10:	IF ip_state = BYTE#3 THEN (* Bei IP_Control anmelden *)
		url_length := LEN(domain_copy);
		char_count := 17 + url_length; (* sendebuffer initialisieren *)
		FOR i := 0 TO char_count DO
			S_BUF.BUFFER[i] := BYTE#00;
		END_FOR;
		tid := UINT_TO_BYTE(BYTE_TO_UINT(tid) + UINT#1);
		S_BUF.BUFFER[01] := tid; (* Transaction ID lowbyte *)
		S_BUF.BUFFER[02] := BYTE#16#01; (* Flags: highbyte *)
		S_BUF.BUFFER[05] := BYTE#16#01; (* Questions: lowbyte *)
		i := url_length + 12;	(* den servernamen von hinten nach vorne bearbeiten *)
		char_count := 0;
		WHILE i > 12 DO
			char := CODE(STR:=domain_copy,POS:=i - 12);
			IF char = BYTE#46 THEN (* prüfe auf haupt/sub domänen namens-teiler "." *)
				S_BUF.BUFFER[i] := INT_TO_BYTE(char_count); (* anstelle des teilers "." wird die länge des erkannten haupt/sub domänennames eingetragen *)
				char_count := 0;
			ELSE
				S_BUF.BUFFER[i] := char; (* char in buffer eintragen *)
				char_count := char_count + 1; (* anzahl char zählen *)
			END_IF;
			i := i - 1;
		END_WHILE;
		S_BUF.BUFFER[i] := INT_TO_BYTE(char_count); (* längenangabe des ganz linken (ersten) domänennamens eintragen *)
		i := url_length + 15; (* position hinter dem servernamen *)
		S_BUF.BUFFER[i] := BYTE#01; (* Type: A Hostaddress lowbyte *)
		i := i + 2;
		S_BUF.BUFFER[i] := BYTE#01; (* Class: IN lowbyte *)
		i := i + 1;
		(* IP Datenverkehr einrichten *)
		IP_C.C_PORT := WORD#53; (* Portnummer eintragen *)
		IP_C.C_IP := IP4_DNS; (* IP eintragen *)
		IP_C.C_MODE := BYTE#1; (* Mode: UDP+AKTIV+PORT+IP *)
		IP_C.C_ENABLE := TRUE; (* Verbindungsaufbau freigeben *)
		IP_C.TIME_RESET := TRUE; (* Zeitueberwachung rücksetzen *)
		IP_C.R_OBSERVE  := TRUE; (* Datenempfang ueberwachen *)
		S_BUF.SIZE := INT_TO_UINT(i); (* sendelänge eintragen *)
		R_BUF.SIZE := UINT#0; (* Empfangslänge rücksetzen *)
		state := 30;

        		(*####################  DEBUG-MESSAGE  ###################################*)
        		(*IF _debug_enable THEN
            		LOG_CL.NEW_MSG := 'DNS: S10 SEND';
            		LOG_MSG();
        		END_IF;*)
        		(*########################################################################*)
	END_IF;

30:	IF IP_C.ERROR <> DWORD#00 THEN
		ERROR := IP_C.ERROR;
		state := 99;
        		(*####################  DEBUG-MESSAGE  ###################################*)
        		(*IF _debug_enable THEN
            		LOG_CL.NEW_MSG := 'DNS: S30 ERROR ~1';
            		LOG_CL.PRINTF[1]  := DWORD_TO_STRING(ERROR);
            		LOG_MSG();
        		END_IF;*)
        		(*########################################################################*)

	ELSIF (S_BUF.SIZE = UINT#0) AND (tid = R_BUF.BUFFER[1]) AND (R_BUF.SIZE >= INT_TO_UINT(34 + url_length)) THEN	(* prüfe ob antwort telegramm die richtige Transaction-ID und mindestlänge hat *)
		ERROR := BYTE_TO_DWORD(R_BUF.BUFFER[3] AND BYTE#2#0000_1111); (* prüfe Return code der Flags. 4 bits *)
		IF ERROR = DWORD#00 THEN
			anc := R_BUF.BUFFER[7]; (* Anzahl der Answer-RR *)
			IP_C.R_OBSERVE := FALSE; (* Datenempfang ueberwachen *)
			state := 40;
		ELSE
			state := 99;
		END_IF;
	END_IF;

40:	IF anc > 0 THEN
		anc := anc - 1;
		WHILE i < R_BUF.SIZE DO
			x := R_BUF.BUFFER[i];
			IF rr_stop = FALSE THEN
				IF x > BYTE#63 THEN (* zeiger auf namen *)
					i := i + 1;
					rr_stop := TRUE;
				ELSIF x= BYTE#0 THEN (* namens ende *)
					rr_stop := TRUE;
				ELSE
					i := i + x; (* namen *)
				END_IF;
				i := i + 1;
			ELSE
				rr_stop := FALSE;
				IF R_BUF.BUFFER[i+1] = BYTE#1 AND R_BUF.BUFFER[i+3] = BYTE#1 THEN (* Type A / Class IN *)
					i := i + 4;
					ttl_tmp := DWORD_OF_BYTE(R_BUF.BUFFER[i],R_BUF.BUFFER[i+1],R_BUF.BUFFER[i+2],R_BUF.BUFFER[i+3]); (* Time to live *)
					i := i + 6;
					IF ttl_tmp >= ttl_last THEN (* TTL ist länger *)
						ttl_last := ttl_tmp;
						IP4 := DWORD_OF_BYTE(R_BUF.BUFFER[i],R_BUF.BUFFER[i+1],R_BUF.BUFFER[i+2],R_BUF.BUFFER[i+3]); (* IP-Adresse *)
					END_IF;
					i := i + 4;
				ELSE
					i := i + 9;
					i := i + R_BUF.BUFFER[i] + 1; (* offset zu nächsten Block *)
				END_IF;
				EXIT;
			END_IF;
		END_WHILE;
	ELSE
		IF ttl_last > DWORD#0 THEN (* gültige RR mit IP gefunden *)
			DONE := TRUE;
            		(*####################  DEBUG-MESSAGE  ###################################*)
            		(*IF _debug_enable THEN
                			LOG_CL.NEW_MSG := 'DNS: S40 OK';
                			LOG_MSG();
            		END_IF;*)
            		(*########################################################################*)
		END_IF;
		state := 99;
	END_IF;

99:	R_BUF.SIZE := UINT#0; (* Empfangslänge rücksetzen *)
	ip_state := BYTE#4; (* Abmelden *)
	state := 00;

END_CASE;

activate_last := ACTIVATE; (* letzten Status sichern zur Flankenerkennung *)
IP_FIFO(FIFO:=IP_C.FIFO,STATE:=ip_state,ID:=ip_id); (* IP_FIFO *)

(* revision history

ks	18. oct. 2008	rev 1.0
	original version

ks	20. oct. 2009	rev 1.1
	unbenutzten code entfernt, all buffer base 0

ks	20. dec. 2010	rev 1.2
	parsing nach rfc1305
*)


(*----------------------------------------------------------------------------------------------------------------*)
(* Flags: 0x0100 (Standard query)                                                                                            *)
(* 0... .... .... .... = Response: Message is a query                                                                   *)
(* .000 0... ....  = Opcode: Standard query (0)                                                                          *)
(* .... ..0. .... .... = Truncated: Message is not truncated                                                          *)
(* .... ...1 .... .... = Recursion desired: Do query recursively                                                    *)
(* .... .... .0.. .... = Z: reserved (0)                                                                                                  *)
(* .... .... ...0 .... = Non-authenticated data OK: Non-authenticated data is unacceptable *)
(*-----------------------------------------------------------------------------------------------------------------*)

(*      0  1  2  3  4  5  6  7  8  9  0  1  2  3  4  5  *)
(*    +--+--+--+--+--+--+--+--+--+--+--+--+--+--+--+--+ *)
(*    |                      ID                       | idx: 0/1   *)
(*    +--+--+--+--+--+--+--+--+--+--+--+--+--+--+--+--+ *)
(*    |QR|   Opcode  |AA|TC|RD|RA|   Z    |   RCODE   | idx: 2/3   *)
(*    +--+--+--+--+--+--+--+--+--+--+--+--+--+--+--+--+ *)
(*    |                    QDCOUNT                    | idx: 4/5   *)
(*    +--+--+--+--+--+--+--+--+--+--+--+--+--+--+--+--+ *)
(*    |                    ANCOUNT                    | idx: 6/7   *)
(*    +--+--+--+--+--+--+--+--+--+--+--+--+--+--+--+--+ *)
(*    |                    NSCOUNT                    | idx: 8/9   *)
(*    +--+--+--+--+--+--+--+--+--+--+--+--+--+--+--+--+ *)
(*    |                    ARCOUNT                    | idx: 10/11 *)
(*    +--+--+--+--+--+--+--+--+--+--+--+--+--+--+--+--+ *)

(*
Errorcodes  Description	References 
000	No error. 		 	The request completed successfully.
001	Format error. 		The name server was unable to interpret the query. 
002	Server failure.  	The name server was unable to process this query due to a problem with the name server. 
003	Name Error. 	 	Meaningful only for responses from an authoritative name server, this code signifies that the domain name referenced in the query does not exist.
004	Not Implemented. 	The name server does not support the requested kind of query.
005	Refused. 			The name server refuses to perform the specified operation for policy reasons.
  						 For example, a name server may not wish to provide the information to the particular requester, or a name server may not wish to perform a particular operation (e.g., zone transfer) for particular data.
006	YXDomain.			Name Exists when it should not. 
007	YXRRSet. RR			Set Exists when it should not. 
008	NXRRSet. RR			Set that should exist does not. 
009	NotAuth.			Server Not Authoritative for zone. 
010	NotZone,			Name not contained in zone. 
255	Timeout				No Response  
   

beispiel einer DNS Request von google.at
ein request mit 3 Answer-Blocks


Domain Name System (response)
[Request In: 3]
[Time: 0.027533000 seconds]
Transaction ID: 0x5e1a
Flags: 0x8180 (Standard query response, No error)
1... .... .... .... = Response: Message is a response
.000 0... .... .... = Opcode: Standard query (0)
.... .0.. .... .... = Authoritative: Server is not an authority for domain
.... ..0. .... .... = Truncated: Message is not truncated
.... ...1 .... .... = Recursion desired: Do query recursively
.... .... 1... .... = Recursion available: Server can do recursive queries
.... .... .0.. .... = Z: reserved (0)
.... .... ..0. .... = Answer authenticated: Answer/authority portion was not authenticated
.... .... .... 0000 = Reply code: No error (0)
Questions: 1
Answer RRs: 3
Authority RRs: 0
Additional RRs: 0

Queries
google.at: type A, class IN
Name: google.at
Type: A (Host address)
Class: IN (0x0001)

Answers
google.at: type A, class IN, addr 72.14.221.104
Name: google.at
Type: A (Host address)
Class: IN (0x0001)
Time to live: 19 minutes, 9 seconds
Data length: 4
Addr: 72.14.221.104

google.at: type A, class IN, addr 66.249.93.104
Name: google.at
Type: A (Host address)
Class: IN (0x0001)
Time to live: 19 minutes, 9 seconds
Data length: 4
Addr: 66.249.93.104

google.at: type A, class IN, addr 216.239.59.104
Name: google.at
Type: A (Host address)
Class: IN (0x0001)
Time to live: 19 minutes, 9 seconds
Data length: 4
Addr: 216.239.59.104
*)
END_FUNCTION_BLOCK

(* POU IP_FIFO, ST *)
FUNCTION_BLOCK IP_FIFO
VAR_IN_OUT
	FIFO : IP_FIFO_DATA;
	ID : BYTE;
	STATE : BYTE;
END_VAR
VAR
	tmp : INT;

	(*LOG_MSG : LOG_MSG;
	_debug_enable : BOOL := TRUE;*)

END_VAR

(*	version 1.0	18. oct. 2008
	programmer 	ks
	tested BY		ks

	IP_FIFO ist ein Zusatzbaustein füR die Zugriffsverwaltung auf IP_CONTROL
*)
IF NOT FIFO.INIT THEN
	FIFO.INIT := TRUE;
	FIFO.NW := 1;
	FIFO.NR := 1;
	FIFO.EMPTY := TRUE;
	FIFO.FULL := FALSE;
	FIFO.TOP := 128; (* Arraygroesse 1 bis x *)
	FIFO.MAX_ID := BYTE#1; (* maximale anzahl von Anmeldungen einer ID *)
END_IF;

(* wenn keine ID vorhanden dann die naechste freie ID zuteilen *)
IF ID = BYTE#00 THEN
	IF FIFO.ID < INT_TO_BYTE(FIFO.TOP) THEN
		ID := USINT_TO_BYTE(BYTE_TO_USINT(FIFO.ID) + USINT#1); (* ID +1 *)
		FIFO.ID := ID; (* ID eintragen *)
	    	(*####################  DEBUG-MESSAGE  ###################################*)
	    	(*IF _debug_enable THEN
	      		LOG_CL.NEW_MSG := 'FIFO: NEW ID:~1';
	      		LOG_CL.PRINTF[1]  := BYTE_TO_STRING(ID);
	      		LOG_MSG();
	    	END_IF;*)
	    	(*########################################################################*)
	ELSIF STATE < BYTE#200 THEN
		(*####################  DEBUG-MESSAGE  ###################################*)
		(*IF _debug_enable THEN
			LOG_CL.NEW_MSG := 'FIFO: OVERFLOW ADD ID';
			LOG_MSG();
		END_IF;*)
		(*########################################################################*)

		(* sollte nie passieren ! -> es sind zuviele teilnehmer angemeldet *)
		(* es wird keine Nummer vergeben und alle anfragen werden negativ beantwortet *)
		STATE := BYTE#255;
		RETURN;
	END_IF;
END_IF;

IF STATE = BYTE#1 AND NOT FIFO.FULL THEN (* Anmelden *)
	(* nur eintragen wenn maximale anzahl nicht ueberschritten wurde *)
	tmp := BYTE_TO_INT(ID);
	IF FIFO.Y[tmp] < FIFO.MAX_ID THEN
		FIFO.Y[tmp] := USINT_TO_BYTE(BYTE_TO_USINT(FIFO.Y[tmp]) + USINT#1); (* IP_ID Zähler +1 *)
		tmp := FIFO.NW; (* geht bei mir leider nicht anders *)
		FIFO.X[tmp] := ID;
		IF FIFO.NW = FIFO.TOP THEN FIFO.NW := 1; ELSE FIFO.NW := FIFO.NW + 1; END_IF;
		FIFO.FULL := FIFO.NW = FIFO.NR;
		FIFO.EMPTY := FALSE;
		STATE := BYTE#2; (* weiterschalten auf "Warten auf Freigabe" *)
		(*####################  DEBUG-MESSAGE  ###################################*)
		(*IF _debug_enable THEN
			LOG_CL.NEW_MSG := 'FIFO: ADD ID:~1';
			LOG_CL.PRINTF[1]  := BYTE_TO_STRING(ID);
			LOG_MSG();
		END_IF;*)
		(*########################################################################*)

	END_IF;
END_IF;

IF STATE = BYTE#2 AND NOT FIFO.EMPTY THEN (* check current stack element *)
	tmp := FIFO.NR; (* geht bei mir leider nicht anders *)
	IF ID = FIFO.X[tmp] THEN
	STATE := BYTE#3; (* weiterschalten auf "Zugriffsfreigabe" *)
	END_IF;
END_IF;

IF STATE = BYTE#4 AND NOT FIFO.EMPTY THEN (* remove from stack *)
	tmp := FIFO.NR; (* geht bei mir leider nicht anders *)
	IF ID = FIFO.X[tmp] THEN
		tmp := BYTE_TO_INT(ID); (* geht bei mir leider nicht anders *)
		FIFO.Y[tmp] := USINT_TO_BYTE(BYTE_TO_USINT(FIFO.Y[tmp]) - USINT#1); (* ID Zähler -1 *)
		IF FIFO.NR = FIFO.TOP THEN FIFO.NR := 1; ELSE FIFO.NR := FIFO.NR + 1; END_IF;
		FIFO.EMPTY := FIFO.NR = FIFO.NW;
		FIFO.FULL := FALSE;
		(*####################  DEBUG-MESSAGE  ###################################*)
		(*IF _debug_enable THEN
			LOG_CL.NEW_MSG := 'FIFO: REMOVE ID:~1';
			LOG_CL.PRINTF[1]  := BYTE_TO_STRING(ID);
			LOG_MSG();
		END_IF;*)
		(*########################################################################*)
	END_IF;
	STATE := BYTE#5; (* "Remove done" *)
END_IF;

(* revision history
ks	18. oct. 2008	rev 1.0
	original version

*)
END_FUNCTION_BLOCK

(* POU IP4_DECODE, ST *)
FUNCTION IP4_DECODE : DWORD
VAR_INPUT
	str : STRING(15);
END_VAR
VAR
	pos: INT;
END_VAR

(*
version 1.1	10. mar 2009
programmer 	kurt
tested by		hugo

IP4_DECODE testet ob ein string eine gültige IPv4 Adresse enthält und gibt die 4 Bytes der IP Adresse als DWORD zurück.

*)
pos := FIND(str, '.');
WHILE pos > 0 DO
	IP4_DECODE := SHL(IP4_DECODE,8) OR STRING_TO_DWORD(LEFT(str,pos - 1));
	str := DELETE(str, pos, 1);
	pos := FIND(str, '.');
END_WHILE;
IP4_DECODE := SHL(IP4_DECODE,8) OR STRING_TO_DWORD(str);


(* revision history
hm		29. feb 2008	rev 1.0
	original version

hm	10. mar. 2009	rev 1.1
	new algorythm
*)
END_FUNCTION

(* POU IP_CONTROL, ST *)
FUNCTION_BLOCK IP_CONTROL
VAR_IN_OUT
	IP_C : IP_C; (* IP_Control Verwaltungsstruktur *)
	S_BUF : NETWORK_BUFFER; (* Externer Sendbuffer *)
	R_BUF : NETWORK_BUFFER; (* Externer Receivebuffer *)
END_VAR
VAR_INPUT
	IP : DWORD; (* IP Adresse *)
	PORT : WORD; (* Port Nummer *)
	TIME_OUT : TIME; (* Ueberwachungszeit Connect / Send / Receive *)
END_VAR
VAR
	c_time : UDINT; (* CONNECT-Time (Zeit bei nicht vorhandener Verbindung) *)
	s_time : UDINT; (* SEND-Time    (Zeit seit letzten Datensenden) *)
	r_time : UDINT; (* RECEIVE-Time (Zeit seit letztem Datenempfang) *)

	c_enable : BOOL; (* Connect: freigabe *)
	c_ip : DWORD; (* Connect: aktuelle IP-Adresse *)
	c_ip_str : STRING(15);
	c_port : WORD; (* Connect: aktuelle Port-Nummer *)
	c_mode : BYTE; (* Connect: aktueller Mode UDP/TCP...... *)
	c_status : BYTE; (* Connect: Status (Errorcode) *)
	c_ready : BOOL; (* Connect: Verbindung aufgebaut *)
	c_ready_old : BOOL; (* Connect: letzter Zustand von c_ready für Flankenauswertung *)

	s_total : INT; (* Send: Gesamtanzahl Bytes zum senden *)
	s_cur_pos : INT; (* Send: aktuelle Sendeposition *)
	s_cur_size : INT; (* Send: aktuelle Sendegroesse *)
	s_max_size : INT; (* Send: maximale Telegrammlänge fuer Senden *)
	s_active : BOOL; (* Send: Daten senden ist aktiv *)
	s_status : BYTE; (* Send: Status (Errorcodes) *)
	s_ip_str : STRING(15);
	s_ip_exist : BOOL;

	r_status : BYTE; (* Receive: Status (Errorcodes) *)
	r_count : INT; (* Receive: Anzahl empfangener Bytes *)
	r_offset : INT; (* Receive: aktuelle Position in externen Receivebuffer *)
	r_max_size : INT; (* Receive: groesse des externen Empfangbuffers*)

	new_connection : BOOL; (* Neue Verbindungsparameter vorhanden *)
	tx : DWORD; (* letzter zeitwert *)
	error_time : DWORD; (* aktueller Timeout-Wert *)

	state: BYTE; (* schrittmerker für connect *)
	bytes_received : DINT;
	udp_mode : BOOL;

	socket : T_HSOCKET;
	server : T_HSOCKET;
	fbCreate	: FB_SocketUdpCreate;
	fbConnect : FB_SocketConnect;
	fbClose : FB_SocketClose;
	fbSendTo : FB_SocketUdpSendTo;
	fbReceiveFrom : FB_SocketUdpReceiveFrom;
	fbSend : FB_SocketSend;
	fbReceive : FB_SocketReceive;
	fbListen : FB_SocketListen;
	fbAccept : FB_SocketAccept;
	nErrId : UDINT;
	Send_Busy : BOOL;
	Send_Error : BOOL;
	Send_ErrId : UDINT;

	IPCR : IP_CONTROL_RESET;

	(*LOG_MSG : LOG_MSG;
	_debug_enable : BOOL := TRUE;
	debug_index : INT;
	debug_ID : INT;
	debug_lasterror : DWORD;
	state_last : INT;
	debug_last_id : INT := 255;*)

END_VAR

VAR CONSTANT
	STOP : BYTE := 0;
	UDP_INIT : BYTE:= 31;
	UDP_INIT_WAIT : BYTE:= 32;
	TC_INIT : BYTE := 51;
	TC_CONNECT : BYTE:= 52;
	TS_INIT : BYTE:= 53;
	TS_LISTEN_WAIT : BYTE:= 54;
	TS_ACCEPT : BYTE:= 55;
	TS_ACCEPT_WAIT : BYTE:= 56;
	C_CLOSE : BYTE := 190;
	C_CLOSE_WAIT : BYTE:= 191;
	C_CLOSE2 : BYTE := 192;
	C_CLOSE_WAIT2 : BYTE:= 193;
	C_WAIT : BYTE := 200;
	C_REC : BYTE := 210;
	C_REC_WAIT : BYTE := 211;
	C_SND : BYTE := 220;
	C_SND_WAIT1 : BYTE := 221;
	C_SND_WAIT2 : BYTE := 222;
END_VAR

(*

version 1.7		30. may. 2011
programmer 		ks
tested by			ks

IP_CONTROL ist ein Wrapper-Baustein um eine Hersteller neutrale Schnittstelle zum Ethernet zu schaffen



TYP 	TCP / UDP 	Aktiv / Passiv 		Port-Nummer erforderlich 	IP-Adresse erforderlich
0 		TCP 		Aktiv 			Ja 						Ja
1 		UDP 		Aktiv 			Ja 						Ja
2 		TCP 		Passiv 			Ja 						Ja (Adresse des aktiven Partners)
3 		UDP 		Passiv 			Ja 						Ja (Adresse des aktiven Partners)
4 		TCP 		Passiv 			Ja 						Nein (beliebiger aktiver Partner wird akzeptiert)
5 		UDP 		Passiv 			Ja 						Nein (beliebiger aktiver Partner wird akzeptiert)

*)
(* Bei PLC reset oder Programm Download werden alle alten Verbindungen geschlossen *)
IPCR();
IF NOT IPCR.READY THEN RETURN; END_IF;

(*####################  DEBUG-MESSAGE  ###################################*)
(*IF _debug_enable THEN
	IF IP_C.FIFO.ID > BYTE#0 THEN (* nur wenn Teilnehmer ID's vorhanden sind *)
		debug_index := IP_C.FIFO.NR;
		debug_ID := BYTE_TO_INT(IP_C.FIFO.X[debug_index]);
	END_IF;
END_IF;*)
(*########################################################################*)

(* read system time *)
tx := T_PLC_MS();

IF IP_C.C_PORT = 0 THEN
	IP_C.C_PORT := PORT; (* uebergebenen PORT durch parametrierten PORT ersetzen *)
END_IF;
IF IP_C.C_IP = 0 AND IP_C.C_MODE < 4 THEN
	IP_C.C_IP := IP; (* uebergebene IP durch paramtrierte IP ersetzen *)
END_IF;

new_connection := c_ip <> IP_C.C_IP OR c_mode <> IP_C.C_MODE OR c_port <> IP_C.C_PORT; (* neue Verbindungs erwünscht ? *)
c_enable := IP_C.C_ENABLE AND NOT new_connection;

IF IP_C.C_ENABLE AND IP_C.ERROR = 0 AND state = STOP THEN (* Freigabe,kein Fehler,kein Socket offen *)
	c_ip   := IP_C.C_IP;
	c_mode := IP_C.C_MODE;
	c_port := IP_C.C_PORT;
	c_ip_str := IP4_TO_STRING(c_ip);
	udp_mode := C_MODE.0; (* Mode 1,3,5 = udp *)

	error_time := TIME_TO_DWORD(MAX(T#200ms,TIME_OUT));
	IP_C.TIME_RESET := TRUE; (* Alle Timer ruecksetzen *)
	r_max_size := SIZEOF(R_BUF.BUFFER);
	s_max_size := SIZEOF(S_BUF.BUFFER);

	IF udp_mode THEN (* Mode: 1,3,5 = UDP CLIENT/SERVER *)
		state := UDP_INIT;
	ELSIF c_mode = 0 THEN (* Mode: 0 = TCP CLIENT *)
		state := TC_INIT;
	ELSE
		state := TS_INIT; (* Mode: 2,4 = TCP SERVER *)
	END_IF;

	IF c_mode < 5 THEN (* Empfänger-IP vorgeben *)
		s_ip_str := c_ip_str;
		s_ip_exist := TRUE;
	ELSE
		s_ip_str := '';
		s_ip_exist := FALSE;
	END_IF;

    	(*####################  DEBUG-MESSAGE  ###################################*)
	(*IF _debug_enable THEN
		LOG_CL.NEW_MSG := 'IP_CON: MODE ~1 / IP ~2 / PORT ~3 /ID ~6';
		LOG_CL.PRINTF[1] := BYTE_TO_STRING(C_MODE);
		LOG_CL.PRINTF[2] := IP4_TO_STRING(c_ip);
		LOG_CL.PRINTF[3] := WORD_TO_STRING(c_port);
		LOG_CL.PRINTF[6] := INT_TO_STRING(debug_ID);
		LOG_MSG();
	END_IF;*)
	(*########################################################################*)

END_IF;

(*####################  DEBUG-MESSAGE  ###################################*)
(*IF  _debug_enable THEN
	IF state <> state_last THEN
		LOG_CL.NEW_MSG := 'IP_STEP ~1 -IP_ID ~6';
		LOG_CL.PRINTF[1] := BYTE_TO_STRING(state);
		LOG_CL.PRINTF[6] := INT_TO_STRING(debug_ID);
		LOG_MSG();
		state_last := state;
	END_IF;
END_IF;*)
(*########################################################################*)

(* ---------------------------------------------- *)

CASE state OF

UDP_INIT: (* UDP_CLIENT + SERVER *)
	(* 1. bei UDP-Client wird als lokalport 0 vorgegeben, damit das System automatisch einen freien lokalen Port sucht
	    2. bei UDP Server muss der gewüschte lokalport verwendet werden *)

	fbCreate(bExecute := FALSE);
	fbCreate(	bExecute := TRUE , sSrvNetId := '', sLocalHost := '', nLocalPort := SEL(c_mode = 1,c_port,0) , tTimeOut := TIME_OUT);
	fbCreate.bExecute := FALSE; (* vorbelegung *)
	state := UDP_INIT_WAIT;

UDP_INIT_WAIT:
	fbCreate();
	IF NOT fbCreate.bBusy THEN
		IF NOT fbCreate.bError THEN
			socket := fbCreate.hSocket;
			c_ready := TRUE; (* Connected *)
			state := C_WAIT;
		ELSE
			c_status := 1; (* FB_SocketUdpCreate failed *)
			nErrId := fbCreate.nErrId;
			state := C_CLOSE;
		END_IF;
	END_IF;

(* ---------------------------------------------- *)
TC_INIT: (* TCP-CLIENT (AKTIV) *)
	fbConnect(bExecute := FALSE);
	fbConnect(bExecute := TRUE, sSrvNetId := '', sRemoteHost := c_ip_str, nRemotePort := c_port, tTimeout := TIME_OUT);
	fbConnect.bExecute := FALSE; (* vorbelegung *)
	state := TC_CONNECT;

(* ---------------------------------------------- *)
TC_CONNECT:
	IF NOT c_enable OR c_status = 255 THEN (* keine freigabe oder connect timeout *)
		state := C_CLOSE;
	END_IF;

	fbConnect();
	IF NOT fbConnect.bBusy THEN
		IF fbConnect.bError THEN
			nErrID := fbConnect.nErrId;
			state :=TC_INIT; (* Nochmals versuchen *)
		ELSE
			socket := fbConnect.hSocket;
			c_ready := TRUE; (* Connected *)
			state := C_WAIT;
		END_IF;
	END_IF;
(* ---------------------------------------------- *)
TS_INIT: (* TCP-SERVER (PASSIV) *)
	fbListen(bExecute := FALSE);
	fbListen(bExecute := TRUE , sSrvNetId:= '' , sLocalHost:= '' , nLocalPort:= c_port , tTimeout:= TIME_OUT);
	fbListen.bExecute := FALSE;
	state := TS_LISTEN_WAIT;
(* ---------------------------------------------- *)
TS_LISTEN_WAIT:
	fbListen();
	IF NOT fbListen.bBusy THEN
		IF fbListen.bError THEN
			c_status := 3; (* FB_SocketListen failed *)
			nErrID := fbListen.nErrId;
			state := C_CLOSE;
		ELSE
			server := fbListen.hListener;
			state := TS_ACCEPT;
		END_IF;
	END_IF;
(* ---------------------------------------------- *)
TS_ACCEPT:
	fbAccept(bExecute := FALSE);
	fbAccept(bExecute := TRUE, sSrvNetId := '', hListener := server, tTimeout := TIME_OUT);
	fbAccept.bExecute := FALSE;
	state := TS_ACCEPT_WAIT;
(* ---------------------------------------------- *)
TS_ACCEPT_WAIT:
	fbAccept();
	IF NOT fbAccept.bBusy THEN

		state := TS_ACCEPT; (* vorbelegung  *)

		IF fbAccept.bError THEN
			c_status := 4; (* FB_SocketAccept failed *)
			nErrID := fbAccept.nErrId;
			state := C_CLOSE;
		ELSE (* no error *)
			IF fbAccept.bAccepted THEN
				socket := fbAccept.hSocket;
				IF socket.remoteAddr.sAddr  <> c_ip_str AND c_mode <> 4 THEN
					state := C_CLOSE; (* Remote ablehnen - Verbindung beenden *)
				ELSE
					state := C_WAIT;
					c_ready := TRUE; (* Connected *)
				END_IF;
			END_IF; (* fbAccept.bAccepted *)
		END_IF; (* NOT fbAccept.bError *)
	END_IF; (*  NOT fbAccept.bBusy *)
(* ---------------------------------------------- *)
C_CLOSE:
	c_ready := FALSE;
	IF socket.handle > 0 THEN
		fbClose(bExecute := FALSE );
		fbClose(bExecute := TRUE, sSrvNetId := '',	hSocket := socket);
		fbClose.bExecute := FALSE;
		state := C_CLOSE_WAIT;
	ELSE
		state:= C_CLOSE2;
	END_IF;

C_CLOSE_WAIT:
	fbClose();
	IF NOT fbClose.bBusy THEN
		socket := TCPADS_NULL_HSOCKET; (* Socket rücksetzen *)
		nErrId:= SEL(fbClose.bError,0,fbClose.nErrId);
		state:= C_CLOSE2;
	END_IF;

C_CLOSE2:
	IF server.handle > 0 THEN
		fbClose(bExecute := FALSE );
		fbClose(bExecute := TRUE, sSrvNetId := '',	hSocket := server);
		fbClose.bExecute := FALSE;
		state := C_CLOSE_WAIT2;
	ELSE
		state:= STOP;
	END_IF;

C_CLOSE_WAIT2:
	fbClose();
	IF NOT fbClose.bBusy THEN
		server := TCPADS_NULL_HSOCKET; (* Socket rücksetzen *)
		nErrId:= SEL(fbClose.bError,0,fbClose.nErrId);
		state:= STOP;
	END_IF;

(* ---------------------------------------------- *)

C_WAIT: (* Warten auf Anforderung für Beenden *)
	IF NOT c_enable OR NOT c_ready THEN
		state:= C_CLOSE;
	ELSIF S_BUF.SIZE > 0 AND IP_C.MAILBOX[2] = 0 AND s_ip_exist THEN
		state:= C_SND;
	ELSIF IP_C.MAILBOX[3] = 0 THEN
		state:= C_REC;
	END_IF;

(* ---------------------------------------------- *)

C_REC: (* Daten empfangen *)
	IF R_BUF.SIZE >= INT_TO_UINT(r_max_size) THEN
		R_BUF.SIZE := UINT#0;
		r_status := 254; (* Empfangsbuffer wegen Überlauf rückgesetzt *)
	END_IF;

	r_offset := SEL(udp_mode,UINT_TO_INT(R_BUF.SIZE),0);
	r_count := r_max_size - r_offset;
	bytes_received := 0;

	IF udp_mode THEN
		fbReceiveFrom(bExecute := FALSE );
		fbReceiveFrom(bExecute:= TRUE, sSrvNetId := '', hSocket:= socket, cbLen := r_count, pDest:= ADR(R_BUF.BUFFER), tTimeout:= TIME_OUT);
		fbReceiveFrom.bExecute := FALSE; (* Vorbelegung *)
	ELSE
		fbReceive(bExecute:= FALSE);
		fbReceive(bExecute:= TRUE, sSrvNetId := '' , hSocket:= socket , cbLen:= r_count, pDest:= ADR(R_BUF.BUFFER[r_offset]) , tTimeout:= TIME_OUT);
		fbReceive.bExecute:= FALSE;
	END_IF;
	state := C_REC_WAIT;

C_REC_WAIT:
	IF udp_mode THEN
		fbReceiveFrom(); (* UDP Mode *)
		IF NOT fbReceiveFrom.bBusy THEN
			IF NOT fbReceiveFrom.bError THEN
				IF fbReceiveFrom.nRecBytes > 0 THEN
					IF c_mode <> BYTE#5 AND fbReceiveFrom.sRemoteHost  <> c_ip_str THEN
						R_BUF.SIZE := UINT#0;
					ELSE
						bytes_received := fbReceiveFrom.nRecBytes;
						IF NOT s_ip_exist THEN
							s_ip_str := fbReceiveFrom.sRemoteHost;
							s_ip_exist := TRUE;
						END_IF;
					END_IF;
				END_IF;
				state := C_WAIT;
			ELSIF fbReceiveFrom.nErrId = 16#80072746 THEN (* Verbindung vom Remote beendet *)
				c_status := 253;
				c_ready := FALSE;
				state := C_WAIT;
			ELSE
				nErrId := fbReceiveFrom.nErrId;
				state := C_WAIT;
			END_IF;
		END_IF;
	ELSE
		fbReceive(); (* TCP Mode *)
		IF NOT fbReceive.bBusy THEN
			IF NOT fbReceive.bError THEN
				IF fbReceive.nRecBytes > 0 THEN
					bytes_received := fbReceive.nRecBytes;
				END_IF;
			ELSIF fbReceive.nErrId = 16#8004 THEN (* Verbindung vom Remote beendet *)
				c_status := 253;
				c_ready := FALSE;
			ELSE
				nErrId := fbReceive.nErrId;
			END_IF;
			state := C_WAIT;
		END_IF;
	END_IF;

	IF bytes_received > 0 THEN
		r_time := tx; (* Receive Timer ruecksetzen *)
		R_BUF.SIZE := INT_TO_UINT(r_offset + DINT_TO_UINT(bytes_received)); (* aktuelle buffersize eintragen *)
		IP_C.MAILBOX[1] := IP_C.MAILBOX[1] + 1; (* Receive Info *)
		IF IP_C.MAILBOX[1] = 0 THEN IP_C.MAILBOX[1] := 1; END_IF;
    		(*####################  DEBUG-MESSAGE  ###################################*)
		(*IF _debug_enable THEN
			LOG_CL.NEW_MSG := 'IP_REC DATA: POS: ~1 : SIZE: ~2 TOTAL ~3 -IP_ID ~6';
			LOG_CL.PRINTF[1] := INT_TO_STRING(r_offset);
			LOG_CL.PRINTF[2] := INT_TO_STRING(r_count);
			LOG_CL.PRINTF[3] := UINT_TO_STRING(R_BUF.SIZE);
			LOG_CL.PRINTF[6] := INT_TO_STRING(debug_ID);
			LOG_MSG();
		END_IF;*)
		(*########################################################################*)
	END_IF;

(* ---------------------------------------------- *)
C_SND:
	IF S_BUF.SIZE > 0 THEN
		IF c_ready AND c_enable THEN
			IF NOT s_active THEN
				s_total := LIMIT(0,UINT_TO_INT(S_BUF.SIZE),r_max_size); (* Gesamtanzahl an Bytes limitieren und uebergeben *)
				s_cur_pos  := 0;
				s_cur_size := 0;
				s_active := TRUE; (* Sende-Betrieb aktivieren *)
			END_IF;

			s_cur_pos := s_cur_pos + s_cur_size; (* neue Sende-Datenposition bestimmen *)
			IF s_total > s_cur_pos THEN (* weitere Daten zum senden vorhanden ? *)
				s_cur_size := s_total - s_cur_pos;
				s_cur_size := LIMIT(0, s_cur_size, s_max_size); (* Telegrammlänge begrenzen *)
				s_time := tx; (* Send Timer ruecksetzen *)
				r_time := tx; (* Receive Timer ruecksetzen *)
				state := C_SND_WAIT1;
			ELSE (* keine weitere Sendedaten vorhanden -> Senden beenden *)
				s_active := FALSE;
				S_BUF.SIZE := 0;
				state := C_WAIT;
			END_IF;
		END_IF;
	END_IF;

C_SND_WAIT1:
	IF udp_mode THEN
		fbSendTo(bExecute := FALSE );
		fbSendTo(bExecute := TRUE, sSrvNetId := '', hSocket := socket , cbLen := s_cur_size, pSrc := ADR(S_BUF.BUFFER[s_cur_pos]), sRemoteHost := s_ip_str, nRemotePort := c_port, tTimeout:= TIME_OUT);
		fbSendTo.bExecute := FALSE;
	ELSE
		fbSend(bExecute := FALSE);
		fbSend(bExecute := TRUE, sSrvNetId := '', hSocket := socket , cbLen:= s_cur_size, pSrc:=ADR(S_BUF.BUFFER[s_cur_pos]), tTimeout:= TIME_OUT);
		fbSend.bExecute := FALSE;
	END_IF;
	state := C_SND_WAIT2;

C_SND_WAIT2:
	IF udp_mode THEN
		fbSendTo();
		Send_Busy := fbSendTo.bBusy;
		Send_Error := fbSendTo.bError;
		Send_ErrId := fbSendTo.nErrId;
	ELSE
		fbSend();
		Send_Busy := fbSend.bBusy;
		Send_Error := fbSend.bError;
		Send_ErrId := fbSend.nErrId;
	END_IF;

	IF NOT Send_Busy THEN
		IF NOT Send_Error THEN
    			(*####################  DEBUG-MESSAGE  ###################################*)
			(*IF _debug_enable THEN
				LOG_CL.NEW_MSG := 'IP_SEN SEND_COUNT ~1 -IP_ID ~6';
				LOG_CL.PRINTF[1] := DINT_TO_STRING(s_cur_size);
				LOG_CL.PRINTF[6] := INT_TO_STRING(debug_ID);
				LOG_MSG();
			END_IF;*)
			(*########################################################################*)
			state := C_SND;
		ELSE
			nErrId := Send_ErrId;
			state := C_WAIT;
    			(*####################  DEBUG-MESSAGE  ###################################*)
			(*IF _debug_enable THEN
				LOG_CL.NEW_MSG := 'IP_SEN SEND ERROR ~1 -IP_ID ~6';
				LOG_CL.PRINTF[1] := UDINT_TO_STRING(nErrId);
				LOG_CL.PRINTF[6] := INT_TO_STRING(debug_ID);
				LOG_MSG();
			END_IF;*)
			(*########################################################################*)
		END_IF;
	END_IF;

END_CASE;

(* ---------------------------------------------- *)

IF c_ready THEN
	IF NOT c_ready_old THEN (* Verbindung aufgebaut - positive Flanke erkannt *)
		IP_C.C_STATE := 254;
		IP_C.TIME_RESET := TRUE; (* Alle Timer ruecksetzen *)
    		(*####################  DEBUG-MESSAGE  ###################################*)
		(*IF _debug_enable THEN
			LOG_CL.NEW_MSG := 'IP_CON: CONNECTED -IP_ID ~6';
			LOG_CL.PRINTF[6] := INT_TO_STRING(debug_ID);
			LOG_MSG();
		END_IF;*)
		(*########################################################################*)
	ELSE
		IP_C.C_STATE := 255; (* Verbindung ist aufgebaut *)
	END_IF;
ELSE
	IF c_ready_old THEN (* Verbindung abgebaut - negative Flanke erkannt *)
		IP_C.C_STATE := 1;
		IP_C.MAILBOX[1] := 0; (* Receive Info rücksetzen *)
		IP_C.MAILBOX[2] := 0; (* Send-Pause rücksetzen *)
		IP_C.MAILBOX[3] := 0; (* Receive-Pause rücksetzen *)
		IF NOT new_connection THEN
			s_active := FALSE; (* Sendeaktivitäten stoppen *)
			S_BUF.SIZE := 0; (* Sendelänge löschen *)
			(*IP_C.TIME_RESET := TRUE; *) (* Alle Timer ruecksetzen *)
		END_IF;
    		(*####################  DEBUG-MESSAGE  ###################################*)
		(*IF _debug_enable THEN
			LOG_CL.NEW_MSG := 'IP_CON: DISCONNECTED';
			LOG_MSG();
		END_IF;*)
		(*########################################################################*)

	ELSE
		IP_C.C_STATE := 0; (* Verbindung ist abgebaut *)
	END_IF;
END_IF;

c_ready_old := c_ready;

(* ---------------------------------------------- *)

IF IP_C.TIME_RESET THEN (* Alle Timer ruecksetzen *)
	IP_C.TIME_RESET := FALSE; (* Reset rücksetzen *)
	c_time := tx; (* Connect Timer ruecksetzen *)
	s_time := tx; (* Send Timer ruecksetzen *)
	r_time := tx; (* Receive Timer ruecksetzen *)

	c_status := BYTE#0; (* letzten Connect Fehler rücksetzen *)
	s_status := BYTE#0; (* letzten Send Fehler rücksetzen *)
	r_status := BYTE#0; (* letzten Receive Fehler rücksetzen *)
END_IF;

IF IP_C.R_OBSERVE = FALSE THEN
    r_time := tx;
END_IF;

IF c_status = 0 AND tx - c_time > error_time AND c_enable AND NOT c_ready AND c_mode < 2 THEN (* Connect Timeout *)
	c_status := 255; (* Timeout-Fehler ausgeben *)
END_IF;
IF s_status = 0 AND tx - s_time > error_time AND s_active THEN (* Send Timeout *)
	s_status := 255; (* Timeout-Fehler ausgeben *)
END_IF;
IF r_status = 0 AND tx - r_time > error_time AND c_ready AND IP_C.R_OBSERVE THEN (* Receive Timeout *)
	r_status := 255; (* Timeout-Fehler ausgeben *)
END_IF;

IP_C.ERROR := DWORD_OF_BYTE(c_status,s_status,r_status,0);

(*####################  DEBUG-MESSAGE  ###################################*)
(*IF  _debug_enable THEN
	IF (IP_C.ERROR <> debug_lasterror) THEN
		LOG_CL.NEW_MSG := 'IP_ERROR ~1 -IP_ID ~6';
		LOG_CL.PRINTF[1] := DWORD_TO_STRING(IP_C.ERROR);
		LOG_CL.PRINTF[6] := INT_TO_STRING(debug_ID);
		LOG_MSG();

		debug_lasterror := IP_C.ERROR;
		debug_last_id := debug_ID;
	END_IF;
END_IF;*)
(*########################################################################*)

(* revision history
ks	18. oct. 2008	rev 1.0
	original version
ks	05. jan. 2009	rev 1.1
	zusätzlichen Parameter "Port" hinzugefügt, und Code bei Verbindungsaufbau angepasst
ks	28. feb. 2009	rev 1.2
	connect code angepasst und verkürzung der zyklen bei Send
ks	20. oct. 2009	rev 1.3
	network_buffer basis 0
ks	06. dec. 2009	rev 1.4
	receive_count MAILBOX[1]
ks	10. nov. 2010	rev 1.5
	send_pause MAILBOX[2] and receive_pause MAILBOX[3] 
ks	07. feb. 2011	rev 1.6
	Fehlercode 253 bei Remote-Verbindungsabbruch 
ks	30. may. 2011	rev 1.7
	Fehler bei Empfangsüberwachung
*)
END_FUNCTION_BLOCK

(* POU IP_CONTROL_RESET, ST *)
FUNCTION_BLOCK IP_CONTROL_RESET
VAR_INPUT
END_VAR
VAR_OUTPUT
	READY : BOOL;
END_VAR
VAR
	fbSocketCloseAll : FB_SocketCloseAll;
	step : BYTE;
END_VAR
(* On PLC reset or program download close all old connections *)

CASE TCP_SERVER_RESET OF

2:	READY := TRUE;
	RETURN;

1:	IF step = 0 THEN
		RETURN;
	END_IF;

0:	TCP_SERVER_RESET := 1; (* Reset ist aktiv *)
	step := 1;

END_CASE;

CASE step OF

0:	RETURN;

1:	fbSocketCloseAll(sSrvNetId:= '', bExecute:= TRUE, tTimeout:= T#10s );
	step := 2;

2:	fbSocketCloseAll(bExecute:= FALSE);
	IF fbSocketCloseAll.bBusy = FALSE THEN
		step := 0;
		TCP_SERVER_RESET := 2; (* Reset durchgeführt , Bereit zur Verwendung *)
	END_IF;

END_CASE;
END_FUNCTION_BLOCK

(* POU IP4_TO_STRING, ST *)
FUNCTION IP4_TO_STRING : STRING(15)
VAR_INPUT
	IP4 : DWORD;
END_VAR
VAR
	tmp : STRING(3);
END_VAR

(*
version 1.1	10. mar. 2009
programmer 	kurt
tested by	hugo

IP4_TO_STRING erzeugt eine IP Adresse als String aus einem DWORD..

*)
(* mask bits AND INSERT AT given position *)
tmp := BYTE_TO_STRING(DWORD_TO_BYTE(IP4));
IP4_TO_STRING := CONCAT('...', tmp);
tmp := BYTE_TO_STRING(DWORD_TO_BYTE(SHR(IP4,8)));
IP4_TO_STRING := INSERT(IP4_TO_STRING, tmp, 2);
tmp := BYTE_TO_STRING(DWORD_TO_BYTE(SHR(IP4,16)));
IP4_TO_STRING := INSERT(IP4_TO_STRING, tmp, 1);
tmp := BYTE_TO_STRING(DWORD_TO_BYTE(SHR(IP4,24)));
IP4_TO_STRING := CONCAT(tmp, IP4_TO_STRING);



(* revision history
hm	22. apr 2008	rev 1.0
	original version

hm	10. mar. 2009	rev 1.1
	improved code
*)
END_FUNCTION

(* POU STRING_TO_URL, ST *)
FUNCTION STRING_TO_URL : URL
VAR_INPUT
	STR : STRING(STRING_LENGTH);
	DEFAULT_PROTOCOL : STRING(10);
	DEFAULT_PATH : STRING(80);
END_VAR
VAR
	pos: INT;
	pos2: INT;
END_VAR
VAR_TEMP
	x : STRING(STRING_LENGTH);
END_VAR

(*
version 1.1	20. dec. 2010
programmer 	hugo
tested by		oscat

URL splits a unifrom resource locator in its conponents.

*)
(*

http://hans:geheim@www.example.org:80/demo/example.cgi?land=de&stadt=aa#abschnitt1
|       |      |         |         |   |                   |               |
|       |      |         Host      |   Pfad                Query           Anker
|       |      Passwort            Port
|       Benutzer
Protokoll

*)

(* check if string is empty and return empty url *)
IF STR = '' THEN RETURN; END_IF;

(* extract the protocol *)
(* first we check if the optional protocol is specified ending with a :// *)
pos := FIND(STR, '://');
IF pos > 0 THEN
	(* store protocol and restore the rest of url in temp *)
	STRING_TO_URL.PROTOCOL := LEFT(STR, pos - 1);
	x := RIGHT(STR, LEN(STR) - pos - 2);
ELSE
	x := STR;
	STRING_TO_URL.PROTOCOL := DEFAULT_PROTOCOL;
END_IF;

(* extract user and password if present ending with a @ *)
pos := FIND(x, '@');
IF pos > 0 THEN
	(* extract user *)
	pos2 := FIND(x,':')+1;
	IF pos2 > 1 AND pos2 <= pos THEN
		STRING_TO_URL.USER := LEFT(x,pos2 - 2);
		STRING_TO_URL.PASSWORD := MID(x, pos - pos2, pos2);
	ELSE
		STRING_TO_URL.USER := LEFT(x, pos - 2);
		STRING_TO_URL.PASSWORD := '';
	END_IF;
	x := RIGHT(x, LEN(x) - pos);
ELSE
	STRING_TO_URL.USER := '';
	STRING_TO_URL.PASSWORD := '';
END_IF;

(* extract anchor *)
pos := FIND(x, '#');
IF pos > 0 THEN
	STRING_TO_URL.ANCHOR := RIGHT(x, LEN(x) - pos);
	x := LEFT(x, pos - 1);
ELSE
	STRING_TO_URL.ANCHOR := '';
END_IF;

(* extract query  *)
pos := FIND(x, '?');
IF pos > 0 THEN
	STRING_TO_URL.QUERY := RIGHT(x, LEN(x) - pos);
	x := LEFT(x, pos - 1);
ELSE
	STRING_TO_URL.QUERY := '';
END_IF;

(* extract path  *)
pos := FIND(x, '/');
IF pos > 0 THEN
	STRING_TO_URL.PATH := RIGHT(x, LEN(x) - pos + 1);
	x := LEFT(x, pos - 1);
ELSE
	STRING_TO_URL.PATH := DEFAULT_PATH;
END_IF;

(* extract port and leave domain *)
pos := FIND(x, ':');
IF pos > 0 THEN
	STRING_TO_URL.PORT := STRING_TO_WORD(RIGHT(x, LEN(x) - pos));
	STRING_TO_URL.DOMAIN := LEFT(x, pos - 1);
ELSE
	STRING_TO_URL.PORT := 0;
	STRING_TO_URL.DOMAIN := x;
END_IF;

(* revision history
hm		18. apr 2008	rev 1.0
	original version

ks		20. dec. 2010	rev 1.1
	stringlength 250 , var x

*)
END_FUNCTION

(* POU FILE_PATH_SPLIT, ST *)
FUNCTION FILE_PATH_SPLIT : BOOL
VAR_INPUT
	FILENAME : STRING(STRING_LENGTH);
END_VAR
VAR_IN_OUT
	X : FILE_PATH_DATA;
END_VAR
VAR
	b : INT;
	c : INT;
	d : STRING(1);
	p1 : INT;
	p2 : INT;
END_VAR

(*
version 1.0		01. jan. 2011
programmer		ks
tested by			ks

FILE_PATH_SPLIT zerlegt einen Dateipfad in einzelne Elemente und legt diese in einer Datenstruktur ab.
*)
X.DRIVE := '';
X.DIRECTORY := '';
X.FILENAME := '';
c := LEN(FILENAME);
IF c = 0 THEN
	FILE_PATH_SPLIT := FALSE;
	RETURN;
END_IF;

FOR b := 1 TO c DO
	d := MID(FILENAME, 1, b);
	IF d = ':' THEN
		p1 := b;
	ELSIF d = '/' OR d = '\' THEN
		p2 := b;
	END_IF;
END_FOR;

IF p1 = 2 THEN
	X.DRIVE := LEFT(FILENAME,p1);
END_IF;

IF p2 > 0 AND p2 > p1 THEN
	X.DIRECTORY := MID(FILENAME,p2 - p1,p1+1); (* len , pos *)
END_IF;

X.FILENAME := RIGHT(FILENAME,c - MAX (p1,p2));
FILE_PATH_SPLIT := TRUE;

(* revision history
ks	01. jan. 2011	rev 1.0
	original version
*)
END_FUNCTION

(* POU ELEMENT_GET, ST *)
FUNCTION ELEMENT_GET : STRING(ELEMENT_LENGTH)
VAR_INPUT
	SEP : BYTE;
	POS : INT;
END_VAR
VAR_IN_OUT
	ELEMENT : STRING(ELEMENT_LENGTH);
END_VAR
VAR
	i : INT := 1;
	o : INT := 1;
	pt : POINTER TO ARRAY[1..ELEMENT_LENGTH] OF BYTE;
	po : POINTER TO ARRAY[1..ELEMENT_LENGTH] OF BYTE;
	cnt: INT;
	c: BYTE;
END_VAR

(*
version 1.0	05. apr. 2011
programmer 	ks
tested by		kst

ELEMENT_GET liefert das element an der stelle pos einer liste.
die liste liegt als string von elementen vor die mit den zeichen SEP separiert sind.

*)
(* load pointers *)
pt := ADR(ELEMENT);
po := ADR(ELEMENT_GET);

(* search for the n-th occurence of a separation character and store position in i *)
WHILE (cnt < pos) AND (i < ELEMENT_LENGTH) AND (pt^[i] > 0) DO
	IF pt^[i] = sep THEN cnt := cnt + 1; END_IF;
	i := i + 1;
END_WHILE;

(* copy the list element to output *)
IF i < ELEMENT_LENGTH THEN c := pt^[i]; END_IF;
WHILE (c <> sep) AND (c > 0) AND (o < ELEMENT_LENGTH) AND (i < ELEMENT_LENGTH) DO
	po^[o] :=pt^[i];
	o := o + 1;
	i := i + 1;
	c := pt^[i];
END_WHILE;

(* terminate the output string *)
po^[o] := 0;

(* revision histroy
ks 05. apr. 2011	rev 1.0
	original release

*)
END_FUNCTION

(* POU DLOG_FILE_CSV_SMTP_DEMO, CFC *)
PROGRAM DLOG_FILE_CSV_SMTP_DEMO
VAR
	RTC_2: RTC_2;
	x : DLOG_DATA;
	DLOG_STORE_FILE_CSV : DLOG_STORE_FILE_CSV;
	CLK_PRG: CLK_PRG;
	cur_dt: DT;
	enable: BOOL;
	rtc_set : BOOL := TRUE;

	trig_t : UDINT := 0;
	trig_m : BOOL;

	x1: DLOG_DT;
	x2 : DLOG_REAL;
	x3 : DLOG_DINT;
	x4 : DLOG_BOOL;
	x5: DLOG_STRING;
	GEN_SIN_1: GEN_SIN;
	COUNT_DR: COUNT_DR;
	error_c: DWORD;
	error_t: BYTE;

	DLOG_FILE_TO_SMTP: DLOG_FILE_TO_SMTP;
	smtp_timeout: TIME := T#30s;
	smtp_error_t: BYTE;
	smtp_error_c: DWORD;
	smtp_busy: BOOL;
	smtp_done: BOOL;
	smtp_dti: DT;
	smtp_dti_offset: INT := 60;
	smtp_server: STRING := '110876022:oscat123456@mail.gmx.net';
	smtp_mailfrom: STRING := 'oscat@gmx.net;Station_01';
	smtp_mailto: STRING(STRING_LENGTH) := 'oscat@gmx.net';
	smtp_subject: STRING := 'Das ist der Betreff';
	smtp_body: STRING(STRING_LENGTH) := 'Das ist der Email-Text';
	smtp_delete: BOOL := TRUE;
	smtp_retry: INT := 0;
	smtp_retry_time: TIME := T#60s;
END_VAR
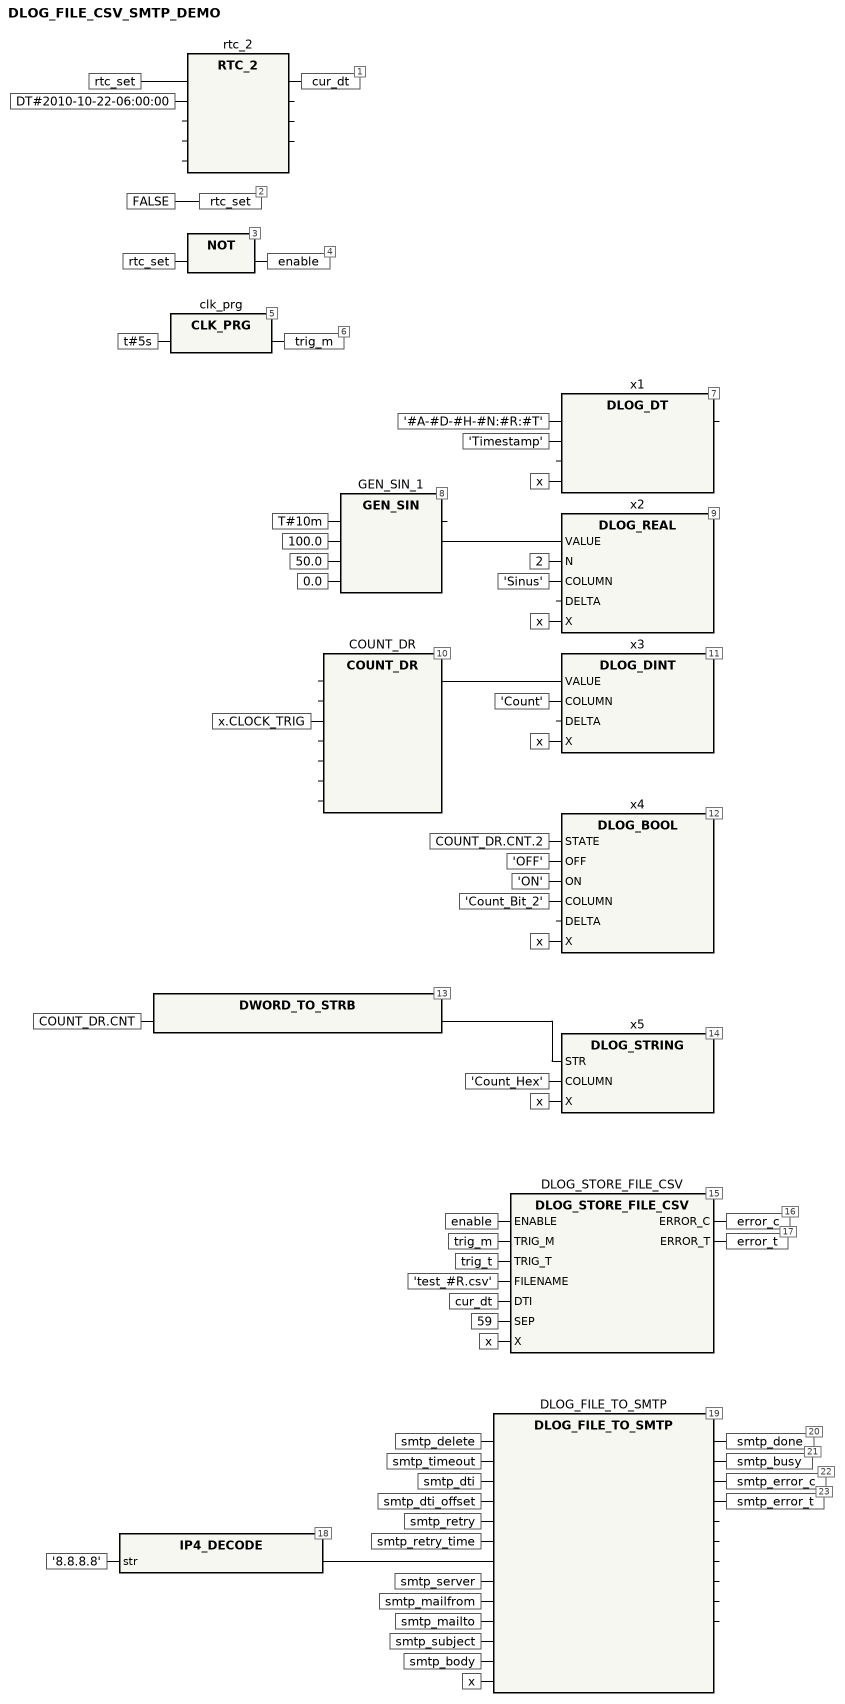
_CFC_ (* Continuous Function Chart, elements in execution order *)
#0 rtc_2:RTC_2(rtc_set, DT#2010-10-22-06:00:00, -, -, -)
#1 cur_dt <= #0.out 1
#2 rtc_set <= FALSE
#3 NOT(rtc_set)
#4 enable <= #3
#5 clk_prg:CLK_PRG(t#5s)
#6 trig_m <= #5
#7 x1:DLOG_DT('#A-#D-#H-#N:#R:#T', 'Timestamp', -, x)
#8 GEN_SIN_1:GEN_SIN(T#10m, 100.0, 50.0, 0.0)
#9 x2:DLOG_REAL(VALUE: #8.out 2, N: 2, COLUMN: 'Sinus', DELTA: -, X: x)
#10 COUNT_DR:COUNT_DR(-, -, x.CLOCK_TRIG, -, -, -, -)
#11 x3:DLOG_DINT(VALUE: #10, COLUMN: 'Count', DELTA: -, X: x)
#12 x4:DLOG_BOOL(STATE: COUNT_DR.CNT.2, OFF: 'OFF', ON: 'ON', COLUMN: 'Count_Bit_2', DELTA: -, X: x)
#13 DWORD_TO_STRB(COUNT_DR.CNT)
#14 x5:DLOG_STRING(STR: #13, COLUMN: 'Count_Hex', X: x)
#15 DLOG_STORE_FILE_CSV:DLOG_STORE_FILE_CSV(ENABLE: enable, TRIG_M: trig_m, TRIG_T: trig_t, FILENAME: 'test_#R.csv', DTI: cur_dt, SEP: 59, X: x)
#16 error_c <= #15.ERROR_C
#17 error_t <= #15.ERROR_T
#18 IP4_DECODE(str: '8.8.8.8')
#19 DLOG_FILE_TO_SMTP:DLOG_FILE_TO_SMTP(smtp_delete, smtp_timeout, smtp_dti, smtp_dti_offset, smtp_retry, smtp_retry_time, #18, smtp_server, smtp_mailfrom, smtp_mailto, smtp_subject, smtp_body, x)
#20 smtp_done <= #19.out 1
#21 smtp_busy <= #19.out 2
#22 smtp_error_c <= #19.out 3
#23 smtp_error_t <= #19.out 4
_END_CFC_
END_PROGRAM

(* POU DLOG_FILE_TO_SMTP, ST *)
(* @OBJECTFLAGS := '0, 8' *)
FUNCTION_BLOCK DLOG_FILE_TO_SMTP
VAR_IN_OUT
	SERVER : STRING;
	MAILFROM : STRING;
	MAILTO : STRING(STRING_LENGTH);
	SUBJECT : STRING;
	BODY : STRING(STRING_LENGTH);
	X : DLOG_DATA;
END_VAR
VAR_INPUT
	FILE_DELETE : BOOL;
	TIMEOUT : TIME := T#30s;
	DTI : DT;
	DTI_OFFSET : INT;
	RETRY : INT;
	RETRY_TIME : TIME := T#30s;
	DNS_IP4 : DWORD;
END_VAR
VAR_OUTPUT
	DONE : BOOL;
	BUSY : BOOL;
	ERROR_C : DWORD;
	ERROR_T : BYTE;
END_VAR
VAR
	UCBD : UNI_CIRCULAR_BUFFER_DATA;
	UCB : UNI_CIRCULAR_BUFFER;
	SMTP_CLIENT : SMTP_CLIENT;
	WT_1 : TON;
	ftrig_old : BOOL;
	files : STRING(STRING_LENGTH);
	step : INT;
	smtp_busy : BOOL;
	smtp_done : BOOL;
	cnt : INT;

	(*LOG_MSG : LOG_MSG;
	_debug_enable : BOOL := TRUE;*)
END_VAR

(*
version 1.1		28. apr. 2011
programmer		ks
tested by			ks

DLOG_FILE_TO_SMTP der Baustein versendet die vom DLOG_STORE_FILE_CSV erzeugten Dateien als Email
*)
(* neue Filenamen speichern *)
IF X.NEW_FILE_RTRIG AND ftrig_old = FALSE THEN
	UCBD.D_HEAD := 1;
	UCBD.D_MODE := 1;
	UCBD.D_STRING := X.NEW_FILE;
	UCB(DATA:=UCBD); (* Daten eintragen *)
END_IF;
ftrig_old := X.NEW_FILE_RTRIG;

CASE step OF

00:	IF UCBD.BUF_COUNT > 0 AND smtp_busy = FALSE THEN
		UCBD.D_MODE := 10; (* Daten lesen *)
		UCB(DATA:=UCBD);
		UCBD.D_MODE := 11; (* Daten löschen *)
		UCB(DATA:=UCBD);
		files := UCBD.D_STRING;
		IF FILE_DELETE THEN
			files := CONCAT(files,';#DEL#');
		END_IF;
		cnt := 0;
		step := 10;
	END_IF;

10:	IF smtp_busy = FALSE THEN
		IF smtp_done THEN
			(*####################  DEBUG-MESSAGE  ###################################*)
			(*IF _debug_enable THEN
				LOG_CL.NEW_MSG := 'F_T_SMTP: /FILE OK >~1<';
				LOG_CL.PRINTF[1] := files;
				LOG_MSG();
			END_IF;*)
			(*########################################################################*)
			step := 0;
		ELSE
			step := 20; (* pause nach error *)
		END_IF;
	END_IF;

20:	IF WT_1.Q THEN (* Wartezeit *)
		cnt := cnt - 1;
		IF RETRY = 0 THEN (* Transfer unbegrenzt wiederholen *)
			(*####################  DEBUG-MESSAGE  ###################################*)
			(*IF _debug_enable THEN
				LOG_CL.NEW_MSG := 'F_T_SMTP: Auftrag unbegrenzt wiederholen /file: ~2';
				LOG_CL.PRINTF[2] := files;
				LOG_MSG();
			END_IF;*)
			(*########################################################################*)
			step := 10; (* Transfer wiederholen *)
		ELSIF cnt >= 0 THEN
			(*####################  DEBUG-MESSAGE  ###################################*)
			(*IF _debug_enable THEN
				LOG_CL.NEW_MSG := 'F_T_SMTP: Auftrag wiederholen /cnt: ~1 /file: ~2';
				LOG_CL.PRINTF[1] := INT_TO_STRING(cnt);
				LOG_CL.PRINTF[2] := files;
				LOG_MSG();
			END_IF;*)
			(*########################################################################*)
			step := 10; (* Transfer wiederholen *)
		ELSE
			(*####################  DEBUG-MESSAGE  ###################################*)
			(*IF _debug_enable THEN
				LOG_CL.NEW_MSG := 'F_T_SMTP: Auftrag verworfen /file: ~2';
				LOG_CL.PRINTF[2] := files;
				LOG_MSG();
			END_IF;*)
			(*########################################################################*)
			step := 0; (* Auftrag verwerfen *)
		END_IF;
	END_IF;

END_CASE;

BUSY := step = 10;
DONE := step = 0;
WT_1(IN:= step = 20, PT:= RETRY_TIME);

SMTP_CLIENT(
	ACTIVATE:= BUSY,
	TIMEOUT:= TIMEOUT,
	DTI:= DTI,
	DTI_OFFSET:= DTI_OFFSET,
	DNS_IP4:= DNS_IP4,
	SERVER:= SERVER,
	MAILFROM:= MAILFROM,
	MAILTO:= MAILTO,
	SUBJECT:= SUBJECT,
	BODY:= BODY,
	FILES:= FILES,
	DONE=> smtp_done,
	BUSY=> smtp_busy,
	ERROR_C=> ERROR_C,
	ERROR_T=> ERROR_T
	);

(* revision history
ks	28. apr. 2011	rev 1.1
	stringfehler bei option 'file_delete'

ks	01. jan. 2011	rev 1.0
	original version
*)
END_FUNCTION_BLOCK

(* POU SMTP_CLIENT, ST *)
FUNCTION_BLOCK SMTP_CLIENT
VAR_INPUT
	ACTIVATE : BOOL;
	TIMEOUT : TIME;
	DTI : DT;
	DTI_OFFSET : INT;
	DNS_IP4 : DWORD;
END_VAR
VAR_OUTPUT
	DONE : BOOL;
	BUSY : BOOL;
	ERROR_C : DWORD;
	ERROR_T : BYTE;
END_VAR
VAR_IN_OUT
	SERVER : STRING;
	MAILFROM : STRING;
	MAILTO : STRING(STRING_LENGTH);
	SUBJECT : STRING;
	BODY : STRING(STRING_LENGTH);
	FILES : STRING(STRING_LENGTH);
END_VAR
VAR
	IP_C : IP_C; (* IP_Control Verwaltungsstruktur *)
	S_BUF : NETWORK_BUFFER;
	R_BUF : NETWORK_BUFFER;
	F_BUF : NETWORK_BUFFER;
	URL_DATA : url;
	DNS_CLIENT : DNS_CLIENT;
	IPC : IP_CONTROL;
	FS : FILE_SERVER;
	FSD : FILE_SERVER_DATA;
	BASE64_ENCODE_STR : BASE64_ENCODE_STR;
	BASE64_ENCODE_STREAM : BASE64_ENCODE_STREAM;
	fpd : FILE_PATH_DATA;
	MD5_CRAM_AUTH : MD5_CRAM_AUTH;
	MD5_RUN : BOOL;
	activate_last : BOOL;
	step : INT;
	snd_step : INT;
	str1 : STRING(STRING_LENGTH);
	str2 : STRING(STRING_LENGTH);
	str3 : STRING;
	snd_text :	STRING(STRING_LENGTH);
	snd_lf_cnt : INT;
	rcv_text :	STRING(STRING_LENGTH);
	rcv_s : STRING(3);
	rcv_state : INT;
	auth_names : STRING := ' PLAIN; LOGIN; CRAM-MD5';
	auth_state : BYTE;
	TON_WAIT : TON;
	last_step : INT;
	next_step : INT;
	timeout2 : TIME;
	timeout3 : TIME;
	last_block : BOOL;
	file_delete : BOOL;
	esmtp : BOOL;
	cnt1 : INT;
	cnt2 : INT;
	cnt3 : INT;
	cnt4 : INT;
	idx1 : INT;
	idx2 : INT;
	idx3 : INT;
	snd_idx : INT;
	snd_enable : BOOL;
	i1 : INT;
	b64_done : BOOL;
	b64_start : BOOL;
	b64_max : UINT := 2880; (* short = 960 / long = 2880 *)
	b64_buf1 : ARRAY [0..47] OF BYTE;
	b64_buf2 : ARRAY [0..63] OF BYTE;
	b64_size1 : INT;
	b64_size2 : INT;
	b64_lf : BOOL;
	b64_str1	: STRING(144);
	b64_str2	: STRING(192);
	md5_user : STRING(64);
	md5_password : STRING(64);
	md5_b64_ts : STRING(64);
	md5_auth_key : STRING(192);
	ip_c_red_disable : BOOL; (* IP_CONTROL - Remote Disconnect Error unterdrücken *)

	(*LOG_MSG : LOG_MSG;
	_debug_enable : BOOL := TRUE;*)
END_VAR

(*
version 1.3		30. may 2011
programmer		ks
tested by			ks

SMTP_CLIENT versendet Email an verschiedene Emailadressen mit optionalen Dateianhängen.



mögliche Rückgabecodes:

Grad der Schwere
 
Die erste Stelle des Rückgabecodes gibt den Grad der Schwere an:
1yz Vorläufige positive Antwort
2yz Antwort über positiven Abschluss 
3yz Positive Zwischenantwort 
4yz Antwort über vorübergehenden negativen Abschluss 
5yz Permanente negative Antwort 
 
Die zweite Stelle gibt die Kategorie der Antwort an: 
x0z Syntaxfehler 
x1z Information 
x2z Verbindung 
x3z Nicht festgelegt 
x4z Nicht festgelegt 
x5z Mail-System 
 
Die dritte Stelle dient zur genaueren Bestimmung der Kategorie. 

Betriebsprotokolle enthalten folgende Codes: 
211 	Systemstatus oder Hilfe-Antwort des Systems  
214 	Hilfe-Nachricht - Informationen zur Verwendung des Empfängers oder zur  
      	Bedeutung eines bestimmten nicht standardmäßigen Befehls; wobei  
      	diese Antwort nur für Personen hilfreich ist, nicht für Systeme 
220 	Service ready (Dienst bereit) 
221 	Service closing transmission channel (Dienst schließt Übertragungskanal) 
235  Authentication succeeded (Authentifizierung erfolgreich)
250 	Requested mail action okay, completed (angeforderte Mail-Maßnahme ok und abgeschlossen) 
251 	User not local; will forward to (Benutzer nicht lokal; Weiterleitung an) 
252 	Cannot VRFY user, but will accept message and attempt delivery (kann Benutzer nicht überprüfen, aber akzeptiert Nachricht und versucht Auslieferung) 
354 	Start mail input; end with. (Mail-Eingabe starten; Ende mit .) 
421 	Service not available, closing transmission channel 	(Dienst nicht verfügbar, Übertragungskanal wird geschlossen) diese Antwort kann auf jeden Befehl folgen, wenn der Dienst weiß, dass er beendet werden muss 
450 	Requested mail action not taken: mailbox unavailable (angeforderte E-Mail-Maßnahme nicht ausgeführt, Mailbox nicht  verfügbar) - z. B. weil Mailbox besetzt 
451	 Requested action aborted: local error in processing (angeforderte Maßnahme abgebrochen: lokaler Fehler bei der Verarbeitung) 
452 	Requested action not taken: insufficient system storage (angeforderte Maßnahme abgebrochen: Systemspeicher nicht ausreichend) 
500 	Syntax error, command unrecognized (Syntaxfehler, Befehl nicht erkannt) - z. B. weil Befehlszeile zu lang 
501 	Syntax error in parameters or arguments (Syntaxfehler in Parametern oder Argumenten) 
502 	Command not implemented (Befehl nicht implementiert) 
504 	Command parameter not implemented (Befehlsparameter nicht implementiert) 
550 	Requested action not taken: mailbox unavailable (Angeforderte Maßnahme nicht ausgeführt: Mailbox nicht verfügbar) 
551 	User not local; please try (Benutzer nicht lokal; versuchen Sie es mit) 
552 	Requested mail action aborted: exceeded storage allocation (angeforderte Mail-Maßnahme abgebrochen: Speicherplatzzuweisung überschritten) 
553 	Requested action not taken: mailbox name not allowed (angeforderte Maßnahme nicht ausgeführt: Mailboxname nicht zulässig) 
554 	Transaction failed (Transaktion fehlgeschlagen) 

#########################
ERROR_T

1 = DNS_CLIENT
2 = SMTP Steuerkanal
4 = FILE_SERVER
5 = Ablaufstörung
#########################

*)
CASE step OF

00:	IF ACTIVATE AND NOT activate_last THEN
		TIMEOUT := MAX(T#10s,TIMEOUT);
		timeout2 := TIMEOUT + T#1s;
		timeout3 := TIMEOUT / 2;
		DONE := FALSE;
		ip_c_red_disable := FALSE;
		ERROR_C := DWORD#0;
		ERROR_T := BYTE#0;
		FSD.ERROR := BYTE#0;
		file_delete := FALSE;
		URL_DATA := STRING_TO_URL(STR:=SERVER,DEFAULT_PROTOCOL:='',DEFAULT_PATH:='/');
		idx1 := FIND(URL_DATA.USER,'%'); (* % Zeichen auf @ ändern *)
		IF idx1 > 0 THEN
			URL_DATA.USER := REPLACE(URL_DATA.USER,'@',1,idx1);
		END_IF;
		esmtp := LEN(URL_DATA.PASSWORD) > 0; (* SMTP oder ExtendedSMTP *)
		step := 10;
	END_IF;

10:	IF DNS_CLIENT.DONE THEN
		step := 20;
	ELSIF DNS_CLIENT.ERROR <> DWORD#0 THEN
		ERROR_C := DNS_CLIENT.ERROR;
		ERROR_T := BYTE#1;
		step := 980;
	END_IF;

20:	(* SMTP Kommunikation einrichten *)
	IP_C.C_PORT := SEL(URL_DATA.PORT = WORD#0,URL_DATA.PORT,WORD#25); (* Portnummer eintragen *)
  	IP_C.C_IP := DNS_CLIENT.IP4; (* IP eintragen *)
  	IP_C.C_MODE := BYTE#0; (* Mode: TCP+ACTIV+PORT *)
  	IP_C.TIME_RESET := TRUE; (* Zeitueberwachung rücksetzen *)
  	IP_C.C_ENABLE := TRUE; (* Verbindungsaufbau freigeben *)
  	IP_C.R_OBSERVE := TRUE; (* Empfangsueberwachung *)
	R_BUF.SIZE := UINT#0;
	snd_enable := TRUE; (* sofortiges senden erlauben *)
	snd_idx := 0;
	step := 30;

30:	IF rcv_state = 220 THEN (* 220 = Service ready *)
		IF esmtp THEN
			snd_text := 'EHLO OSCAT'; (* ExtendedSMTP *)
			next_step := 40;
		ELSE
			snd_text := 'HELO OSCAT'; (* SMTP *)
			next_step := 90;
		END_IF;
		snd_lf_cnt := 1;
	END_IF;

40:	IF rcv_state = 250 THEN (* 250 = Requested mail action okay, completed  *)
		auth_state := BYTE#0;
		str1 := auth_names;
		idx1 := 0;
		idx2 := 1900;
		step := 50;
	END_IF;

50:	str2 := ELEMENT_GET(59, idx1, str1); (* Trennzeichen >;< *)
	IF LEN(str2) > 0 THEN
		IF FIND(rcv_text,str2) > 0 THEN
			auth_state := BIT_LOAD_B(auth_state, TRUE, idx1);
			str3 := str2; (* aktuellen AUTH-Type Namen sichern *)
			idx2 := 1000 + (idx1 * 100); (* Schritt berechnen *)
		END_IF;
		idx1 := idx1 + 1;
	ELSE
		step := 60;
	END_IF;

60:	IF rcv_state = 250 THEN (* 250 = Requested mail action okay, completed  *)
		snd_text := CONCAT('AUTH',str3);
		next_step := idx2; (* mit den jeweiligen Authentifizierung Schritten fortfahren *)
	END_IF;

 (* ++++++++++++++++++++++++++++++++++++++++++++++++++++++*)

90:	IF rcv_state = 235 OR rcv_state = 250 THEN (* 235 = Authentication successful / 250 Requested mail action okay *)
		str2 := MAILFROM;
		str1 := ELEMENT_GET(59, 1, str2);(* Angezeigter Name lesen , Trennzeichen >;< *)
		IF LEN(str1) > 0 THEN
			str3 := INSERT('"" ', str1, 1);
		ELSE
			str3 := '';
		END_IF;
		str1 := ELEMENT_GET(59, 0, str2);(* MAILFROM lesen , Trennzeichen >;< *)
		str2 := INSERT('MAIL FROM: <>', str1, 12);
		snd_text := INSERT(str2, str3, 11);
		str3 := snd_text; (* zur wiederverwendung speichern *)
		next_step := 95;
		cnt1 := ELEMENT_COUNT(35, MAILTO); (* Trennzeichen >#< , Anzahl der Blöcke bestimmen *)
		cnt2 := 0;
	END_IF;

95:	IF rcv_state = 250 THEN (* 250 = Requested mail action okay *)
		IF cnt2 < cnt1 THEN
			str1 := ELEMENT_GET(35, cnt2, MAILTO);(* Trennzeichen >#< *)
			cnt3 := ELEMENT_COUNT(59, str1); (* Trennzeichen >;< , Anzahl der Sub-Blöcke bestimmen *)
			cnt4 := 0;
			cnt2 := cnt2 + 1;
			step := 100; (* Blockinhalt auswerten *)
		ELSE
			step := 110; (* alle Blöcke bearbeitet *)
		END_IF;
	END_IF;

100:	IF rcv_state = 250 THEN (* 250 = Requested mail action okay *)
		IF cnt4 < cnt3 THEN
			str2 := ELEMENT_GET(59, cnt4, str1); (* Trennzeichen >;< *)
			snd_text := INSERT('RCPT TO: <>', str2, 10);
			cnt4 := cnt4 + 1;
			next_step := 100;
		ELSE
			step := 95;
		END_IF;
	END_IF;

110:	IF rcv_state = 250 THEN (* 250 = Requested mail action okay *)
		snd_text := 'DATA';
		next_step := 120;
	END_IF;

120:	IF rcv_state = 354 THEN (* 354 = Start mail input; end with. *)
		snd_enable := FALSE;
		snd_text := REPLACE(str3, 'From', 9, 1); (* 'MAIL FROM' durch "From" ersetzen *)
		cnt2 := 0;
		cnt1 := MIN(2,cnt1); (* BlindCopy Block ausblenden *)
		step := 200;
	END_IF;

200:	IF snd_step = 0 THEN
		IF cnt2 < cnt1 THEN
			str1 := ELEMENT_GET(35, cnt2, MAILTO);(* Trennzeichen >#< *)
			cnt3 := ELEMENT_COUNT(59, str1); (* Trennzeichen >;< , Anzahl der Sub-Blöcke bestimmen *)
			cnt4 := 0;
			cnt2 := cnt2 + 1;
			str3 := SEL(cnt2 = 1,'Cc: <>','To: <>');
			step := 205; (* Blockinhalt auswerten *)
		ELSE
			step := 210; (* alle Blöcke bearbeitet *)
		END_IF;
	END_IF;

205:	IF snd_step = 0 THEN
		IF cnt4 < cnt3 THEN
			str2 := ELEMENT_GET(59, cnt4, str1); (* Trennzeichen >;< *)
			snd_text := INSERT(str3, str2, 5);
			cnt4 := cnt4 + 1;
		ELSE
			step := 200;
		END_IF;
	END_IF;

210:	IF snd_step = 0 THEN
		snd_text := CONCAT('Subject: ',SUBJECT);
		step := 220;
	END_IF;

220:	IF snd_step = 0 THEN
		DTI := UDINT_TO_DT(DT_TO_UDINT(DTI) + INT_TO_UDINT(- DTI_OFFSET * 60)); (* Minuten-Offset auf Sekunden umrechnen und addieren *)
		IF esmtp THEN (* ESMTP Format >Date: Thu, 21 May 1998 05:33:29 -0700< *)
			str2 := ';Mon;Tue;Wed;Thu;Fri;Sat;Sun';
			str1 := ELEMENT_GET(59, DAY_OF_WEEK(DT_TO_DATE(DTI)), str2);
			snd_text := CONCAT('Date: ',str1);
			str1 := DT_TO_STRF(DTI, 0, ', #H #E #A #N:#R:#T +0000', 1);
			snd_text := CONCAT(snd_text,str1);
		ELSE (* SMTP Format >Date: 21 May 98 05:33:29< *)
			snd_text := DT_TO_STRF(DTI, 0, 'Date: #G #E #B #N:#R:#T', 1);
		END_IF;
		step := 230;
	END_IF;

230:	IF snd_step = 0 THEN
		snd_text := 'MIME-Version: 1.0';
		step := 250;
	END_IF;

250:	IF snd_step = 0 THEN
		snd_text := 'Content-Type: multipart/mixed;boundary="x"';
		snd_lf_cnt := 2;
		step := 260;
	END_IF;

260:	IF snd_step = 0 THEN
		snd_enable := TRUE;
		snd_text := 'This is a multi-part message in MIME format.';
		step := 270;
	END_IF;

270:	IF snd_step = 0 THEN
		snd_enable := FALSE;
		snd_text := '--x';
		snd_lf_cnt := 1;
		step := 280;
	END_IF;

280:	IF snd_step = 0 THEN
		snd_text := 'Content-Type: text/plain; format=flowed; charset="iso-8859-1";';
		snd_text := CONCAT(snd_text,' reply-type=original'); (* PCWORX kann nur konstanten mit max 80 zeichen *)
		step := 290;
	END_IF;

290:	IF snd_step = 0 THEN
		snd_text := 'Content-Transfer-Encoding: 8bit';
		snd_lf_cnt := 2;
		step := 300;
	END_IF;

300:	IF snd_step = 0 THEN
		snd_enable := TRUE;
		snd_text := BODY;
		snd_lf_cnt := 2;
		step := 310;
	END_IF;

310:	IF snd_step = 0 THEN
		cnt1 := ELEMENT_COUNT(59, FILES) - 1; (* Anzahl der Dateien *)
		step := 400;
	END_IF;

(* +++++++++++++ File-Attachment ++++++++++++ *)
400:	IF cnt1 >= 0 THEN
		str1 := ELEMENT_GET(59, cnt1, FILES);
		FILE_PATH_SPLIT(FILENAME:=str1,X:=fpd); (* Datei-Path zerlegen *)
		IF fpd.FILENAME = '#DEL#' THEN
			file_delete := TRUE;
		ELSE
			step := 410;
		END_IF;
		cnt1 := cnt1 - 1;
	ELSE
		step := 800;
	END_IF;

410:	IF snd_step = 0 THEN
		snd_enable := FALSE;
		snd_text := '--x';
		snd_lf_cnt := 1;
		step := 420;
	END_IF;

420:	IF snd_step = 0 THEN
		snd_text := 'Content-Transfer-Encoding: BASE64';
		str2 := CONCAT(fpd.FILENAME,'"');
		step := 430;
	END_IF;

430:	IF snd_step = 0 THEN
		snd_text := CONCAT('Content-Type: application/octet-stream; name="',str2);
		step := 440;
	END_IF;

440:	IF snd_step = 0 THEN
		snd_enable := TRUE;
		snd_text := CONCAT('Content-Disposition: attachment; filename="',str2);
		snd_lf_cnt := 2;
		step := 450;
	END_IF;

450:	IF snd_step = 0 THEN
		FSD.FILENAME := str1; (* Dateiname *)
		FSD.OFFSET := UDINT#0; (* Start bei Dateianfang *)
		FSD.AUTO_CLOSE := T#0s; (* kein Auto-Close verwenden *)
		step := 460;
	END_IF;

460:	FSD.MODE := BYTE#1; (* vorhandene Datei zum lesen öffnen *)
	F_BUF.SIZE := b64_max; (* maximale länge einlesen *)
	idx1 := 0;
	idx2 := 0;
	step := 470;

470:	IF FSD.MODE = BYTE#0 AND FSD.ERROR = BYTE#0 THEN
		last_block := FSD.FILE_SIZE = FSD.OFFSET;
		b64_size1 := MIN(48,UINT_TO_INT(F_BUF.SIZE) - idx1);
		IF b64_size1 > 0 THEN
			idx3 := b64_size1 - 1;
			FOR i1 := 0 TO idx3 DO (* daten in BASE64 buffer kopieren *)
				b64_buf1[i1] := F_BUF.BUFFER[idx1];
				idx1 := idx1 + 1;
			END_FOR;
			BASE64_ENCODE_STREAM( SIZE1:= b64_size1, BUF1:= b64_buf1, BUF2:= b64_buf2, SIZE2=> b64_size2); (* BASE64 Kodierung *)
			idx3 := b64_size2 - 1;
			FOR i1 := 0 TO idx3 DO (* Daten aus BASE64 buffer kopieren *)
				S_BUF.BUFFER[idx2] := b64_buf2[i1];
				idx2 := idx2 + 1;
			END_FOR;
			b64_lf := TRUE;
			(*####################  DEBUG-MESSAGE  ###################################*)
			(*IF _debug_enable THEN
				LOG_CL.NEW_MSG := 'B64: FILE ~1 /SIZE ~2 /OFF ~3 /BSIZE ~4 /idx1 ~5 /idx2 ~6';
				LOG_CL.PRINTF[1] := FSD.FILENAME;
				LOG_CL.PRINTF[2] := UDINT_TO_STRING(FSD.FILE_SIZE);
				LOG_CL.PRINTF[3] := UDINT_TO_STRING(FSD.OFFSET);
				LOG_CL.PRINTF[4] := INT_TO_STRING(b64_size1);
				LOG_CL.PRINTF[5] := INT_TO_STRING(idx1);
				LOG_CL.PRINTF[6] := INT_TO_STRING(idx2);
				LOG_MSG();
			END_IF;*)
			(*########################################################################*)
		ELSE
			b64_lf := last_block;
			step := 480; (* block beendet  *)
		END_IF;
		IF b64_lf THEN
			S_BUF.BUFFER[idx2] := BYTE#16#0D;
			idx2 := idx2 + 1;
			S_BUF.BUFFER[idx2] := BYTE#16#0A;
			idx2 := idx2 + 1;
		END_IF;
		(*####################  DEBUG-MESSAGE  ###################################*)
		(*IF _debug_enable THEN
			LOG_CL.NEW_MSG := 'B64: exit ~1 /SIZE ~2 /OFF ~3 /eof ~4 /lf_cnt ~5';
			LOG_CL.PRINTF[1] := FSD.FILENAME;
			LOG_CL.PRINTF[2] := UDINT_TO_STRING(FSD.FILE_SIZE);
			LOG_CL.PRINTF[3] := UDINT_TO_STRING(FSD.OFFSET);
			LOG_CL.PRINTF[4] := BOOL_TO_STRING(last_block);
			LOG_CL.PRINTF[5] := INT_TO_STRING(snd_lf_cnt);
			LOG_MSG();
		END_IF;*)
		(*########################################################################*)
	END_IF;

480:	S_BUF.SIZE := INT_TO_UINT(idx2); (* Daten senden *)
	(*####################  DEBUG-MESSAGE  ###################################*)
	(*IF _debug_enable THEN
		LOG_CL.NEW_MSG := 'B64: tcp_send ~1';
		LOG_CL.PRINTF[1] := INT_TO_STRING(idx2);
		LOG_MSG();
	END_IF;*)
	(*########################################################################*)
	step := 490;

490:	IF S_BUF.SIZE = UINT#0 THEN (* warten bis alle daten gesendet sind *)
		step := SEL(last_block ,460,400);
	END_IF;

(* ++++++++++++++++++++++++++++++++++++++++ *)

800:	IF snd_step = 0 THEN
		snd_enable := FALSE;
		snd_text := '--x--';
		snd_lf_cnt := 2;
		step := 810;
	END_IF;

810:	IF snd_step = 0 THEN
		snd_enable := TRUE;
		snd_text := '.';
		snd_lf_cnt := 1;
		step := 820;
	END_IF;

820:	IF rcv_state = 250 THEN (* 250 = Requested mail action okay *)
		snd_text := 'QUIT';
		ip_c_red_disable := TRUE;
		next_step := 830;
	END_IF;

830:	IF rcv_state = 221  OR TON_WAIT.ET > timeout3 THEN (* 221 = Service closing transmission channel *)
		step := 900;
	END_IF;

(* ================================================== *)

900:IF FILE_DELETE THEN (* Dateien nach transfer löschen *)
		cnt1 := ELEMENT_COUNT(59, FILES) - 1; (* Anzahl der Dateien *)
		step := 910;
	ELSE
		step := 950;
	END_IF;

910:	IF FSD.MODE = BYTE#0 AND FSD.ERROR = BYTE#0 THEN
		IF cnt1 >= 0 THEN
			str1 := ELEMENT_GET(59, cnt1, FILES);
			IF str1 <> '#DEL#' THEN
				FSD.FILENAME := str1;
				FSD.MODE := BYTE#4; (* File Remove *)
			END_IF;
			cnt1 := cnt1 - 1;
		ELSE
			step := 950;
		END_IF;
	END_IF;

950:DONE := TRUE;
	step := 980;

980:IP_C.C_ENABLE := FALSE; (* SMTP Steuerkanal schliessen *)
	S_BUF.SIZE := UINT#0;
	R_BUF.SIZE := UINT#0;
	snd_step := 0;
	next_step := 0;
	FSD.MODE := BYTE#5; (* Datei schliessen *)
	step := 990;

990:IF IP_C.C_STATE = BYTE#0 AND FSD.FILE_OPEN = FALSE THEN
		step := 0;
	END_IF;

(*  +++++++++++++++++ Authentifizierung +++++++++++++++++ *)

(* PLAIN ++++++++++++++++++++++++++++++++++++++++++++++++++++++++++ *)
1000:IF rcv_state = 334 THEN (* 334 = Authentifizierung  *)
		cnt1 := LEN(URL_DATA.USER);
		cnt2 := LEN(URL_DATA.PASSWORD);
		IF cnt1 + cnt2 <= 46 THEN (* USER + PASSWORD dürfen zusammen maximal 46 Zeichen haben *)
			b64_buf1[0] := BYTE#0;
			FOR i1 := 1 TO cnt1 DO
				b64_buf1[i1] := CODE(URL_DATA.USER, i1);
			END_FOR;
			b64_size1 := cnt1 + 1;
			b64_buf1[b64_size1] := BYTE#0;
			b64_size1 := b64_size1 + 1;
			FOR i1 := 1 TO cnt2 DO
				b64_buf1[b64_size1] := CODE(URL_DATA.PASSWORD, i1);
				b64_size1 := b64_size1 + 1;
			END_FOR;
			BASE64_ENCODE_STREAM( SIZE1:= b64_size1, BUF1:= b64_buf1, BUF2:= b64_buf2, SIZE2=> b64_size2); (* BASE64 Kodierung *)
			idx1 := b64_size2 - 1;
			FOR i1 := 0 TO idx1 DO
				S_BUF.BUFFER[i1] := b64_buf2[i1];
			END_FOR;
			S_BUF.BUFFER[b64_size2] := BYTE#16#0D;
			b64_size2 := b64_size2 + 1;
			S_BUF.BUFFER[b64_size2] := BYTE#16#0A;
			b64_size2 := b64_size2 + 1;
			S_BUF.SIZE := INT_TO_UINT(b64_size2);
			rcv_state := 0;
		END_IF;
		step := 90;
	END_IF;

(* LOGIN ++++++++++++++++++++++++++++++++++++++++++++++++++++++++++ *)
1100:IF rcv_state = 334 THEN (* 334 = Authentifizierung  *)
		b64_str1 := URL_DATA.USER;
		b64_start := TRUE; (* BASE64 kodierung von Username *)
		step := 1120;
	END_IF;

1120:IF b64_start AND b64_done THEN
		b64_start := FALSE;
		snd_text := b64_str2;
		next_step := 1130;
	END_IF;

1130:IF rcv_state = 334 THEN (* 334 = Password:  *)
		b64_str1 := URL_DATA.PASSWORD;
		b64_start := TRUE; (* BASE64 kodierung von Password *)
		step := 1140;
	END_IF;

1140:IF b64_start AND b64_done THEN
		b64_start := FALSE;
		snd_text := b64_str2;
		next_step := 90;
	END_IF;

(* CRAM-MD5 (Challenge-Response Authentication Mechanism, Message Digest 5) Authentifizierung auf Basis von MD5-HMAC-Algorithmus. *)
1200:IF rcv_state = 334 THEN (* 334 = Authentifizierung  *)
		md5_b64_ts := RIGHT(rcv_text,LEN(rcv_text) - 4);
		md5_user := URL_DATA.USER;
		md5_password := URL_DATA.PASSWORD;
		MD5_RUN := TRUE;
		step := 1220;
	END_IF;

1220:MD5_CRAM_AUTH(RUN:=MD5_RUN,USERNAME:=md5_user,PASSWORD:=md5_password,B64_TS:=md5_b64_ts,AUTH_KEY:=md5_auth_key);
	IF NOT MD5_RUN THEN
		snd_text := md5_auth_key;
		step := 90;
	END_IF;

(* keine Authentifizierung gefunden +++++++++++++++++++++++++++++++ *)
1900: ; (* Auf Laufzeitfehler warten *)

END_CASE;
(* ++++++++++++++++++++++++++++++++++++++++++++++++++++++++++ *)
IF step >= 30 THEN
	IF R_BUF.SIZE > UINT#0 THEN (* Daten wurden empfangen ? *)
		idx1 := UINT_TO_INT(R_BUF.SIZE);
		REPEAT (* zeilenterminierung erkennen und echtes TEXT-Ende bestimmen *)
			idx1 := idx1 - 1;
		UNTIL idx1 = 0 OR R_BUF.BUFFER[idx1] >= BYTE#32 (* TRUE = EXIT *)
		END_REPEAT;
		FOR i1 := 0 TO idx1 DO (* bei multiline alle CRLF durch >^< ersetzen *)
			IF R_BUF.BUFFER[i1] < BYTE#32 THEN
				R_BUF.BUFFER[i1] := BYTE#94; (* >^< *)
			END_IF;
		END_FOR;
		rcv_text := BUFFER_TO_STRING(PT:=ADR(R_BUF.BUFFER),SIZE:=idx1+1,START:=0,STOP:=STRING_LENGTH-1);
		IF LEN(rcv_text) >= 3 THEN (* Statuscode prüfen und auswerten *)
			rcv_s := LEFT(rcv_text,3);
			IF IS_NUM(STR:=rcv_s) THEN (* enthält nur Zahlen ? *)
				rcv_state := STRING_TO_INT(rcv_s);
			END_IF;
			IP_C.R_OBSERVE := FALSE;
		END_IF;
		R_BUF.SIZE := UINT#0; (* daten löschen *)

		(*####################  DEBUG-MESSAGE  ###################################*)
		(*IF _debug_enable THEN
			LOG_CL.NEW_MSG := 'RCV: >~1<';
			LOG_CL.PRINTF[1] := rcv_text;
			LOG_MSG();
		END_IF;*)
		(*########################################################################*)

	END_IF;
END_IF;

(* automatisches Datensenden *)

CASE snd_step OF

00:	IF LEN(snd_text) > 0 THEN

		(*####################  DEBUG-MESSAGE  ###################################*)
		(*IF _debug_enable THEN
			LOG_CL.NEW_MSG := 'SND: >~1< /lf ~2';
			LOG_CL.PRINTF[1] := snd_text;
			LOG_CL.PRINTF[2] := INT_TO_STRING(snd_lf_cnt);
			LOG_MSG();
		END_IF;*)
		(*########################################################################*)

		_STRING_TO_BUFFER(str:=snd_text,pos:=snd_idx,pt:=ADR(S_BUF.BUFFER),size:=SIZEOF(S_BUF.BUFFER)); (* String in puffer kopieren *)
		snd_idx := snd_idx + LEN(snd_text);
		FOR i1 := 1 TO snd_lf_cnt DO
			S_BUF.BUFFER[snd_idx] := BYTE#16#0D;
			snd_idx := snd_idx + 1;
			S_BUF.BUFFER[snd_idx] := BYTE#16#0A;
			snd_idx := snd_idx + 1;
		END_FOR;
		snd_text := '';
		rcv_state := 9999; (* letzen SMTP Status löschen *)

		IF snd_enable THEN
			S_BUF.SIZE := INT_TO_UINT(snd_idx); (* Sendelänge eintragen *)
			R_BUF.SIZE := UINT#0; (* Empfangsbuffer rücksetzen *)
			IP_C.R_OBSERVE := step <= 120 OR step >= 820;
			snd_idx := 0;
			snd_step := 10;
		END_IF;
	END_IF;

10:	IF S_BUF.SIZE = UINT#0 THEN (* warten bis alle daten gesendet sind *)
		IF next_step <> 0 THEN
			step := next_step;
			next_step := 0;
		END_IF;
		snd_step := 0;
	END_IF;

END_CASE;

(* Globale Fehlerbehandlung für Haupt-Routine *)
IF ERROR_T = BYTE#0 AND step > 20 THEN (* noch kein Fehler gespeichert und Hauptroutine aktiv *)

	IF IP_C.ERROR > DWORD#0 AND IP_C.C_ENABLE AND NOT IP_C.TIME_RESET THEN  (* IP Control 1 *)
		IF ip_c_red_disable = FALSE OR IP_C.ERROR <> DWORD#16#FD000000 THEN
			ERROR_C := IP_C.ERROR;
			ERROR_T := BYTE#2;
			step := 980;
		END_IF;
	END_IF;

	IF FSD.MODE = BYTE#0 THEN
		IF FSD.ERROR > BYTE#0 THEN
			ERROR_C := BYTE_TO_DWORD(FSD.ERROR);
			ERROR_T := BYTE#4; (* Dateizugriff *)
			step := 980;
		END_IF;
	END_IF;
END_IF;

IF TON_WAIT.Q THEN (* Ablaufstörung - Schrittkette *)
	ERROR_C := SHL(INT_TO_DWORD(step),16) OR INT_TO_DWORD(rcv_state); (* aktuellen Schritt und letzten SMTP Status eintragen *)
	ERROR_T := BYTE#5;
	step := 980;
END_IF;

(* ######################################################## *)

DNS_CLIENT(IP_C:=IP_C, S_BUF:=S_BUF, R_BUF:=R_BUF, DOMAIN:=URL_DATA.DOMAIN, IP4_DNS:= DNS_IP4, ACTIVATE:=step=10); (* DNS-Client *)
IPC(IP:= DWORD#0, PORT:= WORD#0 , TIME_OUT:= TIMEOUT, IP_C:= IP_C, S_BUF:= S_BUF, R_BUF:= R_BUF); (* SMTP Steuerkanal *)
FS(FSD:=FSD,PT:=F_BUF); (* FILE_SERVER *)
BASE64_ENCODE_STR(RUN:= b64_start, STR1:= b64_str1, STR2:= b64_str2, DONE=> b64_done); (* BASE64 kodierung *)

TON_WAIT(IN:=step = last_step AND step > 0,PT:=timeout2);
last_step := step;
activate_last := ACTIVATE;
BUSY := step <> 0;

(* revision history
ks	01. jan. 2011	rev 1.0
	original version
ks	06. apr. 2011	rev 1.1
	list_len und list_get durch element_count und element_get ersetzt
ks	11. may 2011	rev 1.2
	ip_control - remote disconnect error ausblenden, und sonderbehandlung für pcworx
ks	30. may. 2011	rev 1.3
	fehler bei empfangsüberwachung
*)
END_FUNCTION_BLOCK

(* POU MD5_CRAM_AUTH, ST *)
FUNCTION_BLOCK MD5_CRAM_AUTH
VAR_IN_OUT
	RUN : BOOL;
	USERNAME : STRING(64);
	PASSWORD : STRING(64);
	B64_TS : STRING(64);  (* Base64 coded ServerTimeStamp *)
	AUTH_KEY : STRING(192);
END_VAR
VAR
	BASE64_DECODE_STR : BASE64_DECODE_STR;
	BASE64_ENCODE_STR : BASE64_ENCODE_STR;
	MD5_STREAM : MD5_STREAM;
	step : INT;
	md5_mode : INT;
	buf : ARRAY [0..63] OF BYTE;
	md5 : ARRAY [0..15] OF BYTE;
	md5_first : ARRAY [0..15] OF BYTE;
	md5_str1 : STRING(64);
	md5_str2 : STRING(64);
	size : UDINT;
	n1 : INT;
	n2 : INT;
	pos : UDINT;
	b64d_run : BOOL;
	b64d_done : BOOL;
	b64e_run : BOOL;
	b64e_done : BOOL;
	str_192 : STRING(192);
	str_144 : STRING(144);
	xpad : BYTE;
	pt : POINTER TO BYTE;
END_VAR

(*
version 1.0		10. may 2010
programmer 	ks
tested by		ks

Der Baustein MD5_CRAM_AUTH (Challenge-Response Authentication Mechanism, Message Digest 5) benutzt
das Authentifizierungsverfahren nach dem Challenge-Response-Prinzip auf der Basis des MD5-HMAC-Algorithmus.
Es wird beispielsweise zur Authentifizierung gegenüber SMTP- oder IMAP-Servern eingesetzt, da es die Übertragung des Passworts im Klartext vermeidet.
Durch dieses Verfahren kann auch über unverschlüsselte Kanäle eine sichere Authentifizierung gegenüber einem Server erfolgen


*)
CASE step OF

0:	IF RUN THEN
		step := 5;
		str_192 := B64_TS;
		b64d_run := TRUE;
	END_IF;

5: IF B64D_DONE THEN (* IPAD Zyklus *)
		b64d_run := FALSE;
		xpad := 16#36;
		md5_str1 := PASSWORD;
		md5_str2 := str_144;
		size := 64 + LEN(md5_str2);
		md5_mode := 1;
		step := 10;
	END_IF;

10: IF md5_mode = 3 THEN (* OPAD Zyklus *)
		md5_first := md5; (* md5 array vom IPAD sichern *)
		xpad := 16#5C;
		size := 64 + 16;
		md5_mode := 1;
		step := 20;
	END_IF;

20: IF md5_mode = 3 THEN
		md5_mode := 0;
		str_144 := CONCAT(USERNAME , ' ');
		str_144 := CONCAT(str_144 , MD5_TO_STRH(md5));
		b64e_run := TRUE;
		step := 30;
	END_IF;

30: IF B64E_DONE THEN
		AUTH_KEY := str_192;
		b64e_run := FALSE;
		RUN := FALSE;
		step := 0; (* alles beendet !! *)
	END_IF;

END_CASE;

(* ----------- md5 -------------- *)
CASE md5_mode OF

1:	n2 := LEN(md5_str1) - 1;
	pt := ADR(md5_str1);
	FOR n1 := 0 TO n2 DO (* string in buf kopieren *)
		buf[n1] := pt^ XOR xpad;
		pt := pt + 1;
	END_FOR;
	FOR n1 := n2 + 1 TO 63 DO (* mit ipad füllen *)
		buf[n1] := xpad;
	END_FOR;

2:	(* Data copy and Calc *)
	IF size > 0 AND pos >= 64 THEN
		IF step = 20 THEN
			FOR n1 := 0 TO 15 DO
				buf[n1] := md5_first[n1];
			END_FOR;
		ELSE
			n2 := LEN(md5_str2) - 1;
			pt := ADR(md5_str2);
			FOR n1 := 0 TO n2 DO (* string in buf kopieren *)
				buf[n1] := pt^;
				pt := pt + 1;
			END_FOR;
		END_IF;
	END_IF;

END_CASE;

IF md5_mode > 0 THEN
	MD5_STREAM(SIZE:=size, MODE:=md5_mode, BUF:=buf, MD5:=md5, POS=>pos);
END_IF;

BASE64_DECODE_STR(RUN:=b64d_run, STR1:=str_192, STR2:=str_144, DONE=>b64d_done);
BASE64_ENCODE_STR(RUN:=b64e_run, STR1:=str_144, STR2:=str_192, DONE=>b64e_done);

(* revision history

hm		10. mai. 2010	rev 1.0
	original version
*)
END_FUNCTION_BLOCK

(* POU MD5_STREAM, ST *)
FUNCTION_BLOCK MD5_STREAM
VAR_IN_OUT
	MODE : INT;
	BUF : ARRAY [0..63] OF BYTE;
	MD5 : ARRAY [0..15] OF BYTE;
	SIZE : UDINT;
END_VAR

VAR_OUTPUT
	POS : UDINT;
END_VAR

VAR
	hash : ARRAY [0..3] OF DWORD;
	a : DWORD;
	b : DWORD;
	c : DWORD;
	d : DWORD;
	end : UDINT;
	block : UDINT;
	x : ARRAY [0..15] OF DWORD;
	n : INT;
	n1 : INT;
	z : INT;
	pad_1 : BOOL;
END_VAR

(*
version 1.0	06. dec. 2009
programmer 	ks
tested BY	ks

MD5_STREAM berechnet den MD5 Hash eines Datenstromes
*)
CASE MODE OF

1:	(* Initialisierung der Hash-Werte *)
	hash[0] := DWORD#16#67452301;
	hash[1] := DWORD#16#EFCDAB89;
	hash[2] := DWORD#16#98BADCFE;
	hash[3] := DWORD#16#10325476;

	block := SHR(SIZE,6) + BOOL_TO_UDINT((UDINT_TO_BYTE(SIZE) AND 16#3F) > 55);
	pad_1 := FALSE;
	POS := 0;
	End := SIZE;
	SIZE := MIN(64,End);
	MODE := 2;

2:	(* Fuell-Bytes anhängen *)
	FOR n := UDINT_TO_INT(SIZE) TO 63 DO
		BUF[n] := 0;
	END_FOR;

	IF SIZE < 64 AND NOT pad_1 THEN
		BUF[SIZE] := 2#1000_0000;
		pad_1 := TRUE;
	END_IF;

	POS := POS + SIZE;
	SIZE := MIN(64,End - POS);

	n := 0;	(* Byte-Array in DWORD-Array umkopieren *)
	FOR n1 := 0 TO 15 DO
		x[n1] := DWORD_OF_BYTE(BUF[n+3],BUF[n+2],BUF[n+1],BUF[n]); (* Little Endian Format *)
		n := n + 4;
	END_FOR;

	IF block = 0 THEN (* am Ende des letzten Blocks die Datenlänge eintragen *)
		x[14] := SHL(UDINT_TO_DWORD(End),3); (* Anzahl Datenbits im Little-Endian Format eintragen *)
		MODE := 3;
	ELSE
		block := block - 1;
	END_IF;

	a := hash[0];
	b := hash[1];
	c := hash[2];
	d := hash[3];

	a := MD5_AUX(1, a, b, c, d, X[00], 07, 16#D76AA478); (* 01 *)
	d := MD5_AUX(1, d, a, b, c, X[01], 12, 16#E8C7B756); (* 02 *)
	c := MD5_AUX(1, c, d, a, b, X[02], 17, 16#242070DB); (* 03 *)
	b := MD5_AUX(1, b, c, d, a, X[03], 22, 16#C1BDCEEE); (* 04 *)
	a := MD5_AUX(1, a, b, c, d, X[04], 07, 16#F57C0FAF); (* 05 *)
	d := MD5_AUX(1, d, a, b, c, X[05], 12, 16#4787C62A); (* 06 *)
	c := MD5_AUX(1, c, d, a, b, X[06], 17, 16#A8304613); (* 07 *)
	b := MD5_AUX(1, b, c, d, a, X[07], 22, 16#FD469501); (* 08 *)
	a := MD5_AUX(1, a, b, c, d, X[08], 07, 16#698098D8); (* 09 *)
	d := MD5_AUX(1, d, a, b, c, X[09], 12, 16#8B44F7AF); (* 10 *)
	c := MD5_AUX(1, c, d, a, b, X[10], 17, 16#FFFF5BB1); (* 11 *)
	b := MD5_AUX(1, b, c, d, a, X[11], 22, 16#895CD7BE); (* 12 *)
	a := MD5_AUX(1, a, b, c, d, X[12], 07, 16#6B901122); (* 13 *)
	d := MD5_AUX(1, d, a, b, c, X[13], 12, 16#FD987193); (* 14 *)
	c := MD5_AUX(1, c, d, a, b, X[14], 17, 16#A679438E); (* 15 *)
	b := MD5_AUX(1, b, c, d, a, X[15], 22, 16#49B40821); (* 16 *)

	a := MD5_AUX(2, a, b, c, d, X[01], 05, 16#F61E2562); (* 17 *)
	d := MD5_AUX(2, d, a, b, c, X[06], 09, 16#C040B340); (* 18 *)
	c := MD5_AUX(2, c, d, a, b, X[11], 14, 16#265E5A51); (* 19 *)
	b := MD5_AUX(2, b, c, d, a, X[00], 20, 16#E9B6C7AA); (* 20 *)
	a := MD5_AUX(2, a, b, c, d, X[05], 05, 16#D62F105D); (* 21 *)
	d := MD5_AUX(2, d, a, b, c, X[10], 09, 16#02441453); (* 22 *)
	c := MD5_AUX(2, c, d, a, b, X[15], 14, 16#D8A1E681); (* 23 *)
	b := MD5_AUX(2, b, c, d, a, X[04], 20, 16#E7D3FBC8); (* 24 *)
	a := MD5_AUX(2, a, b, c, d, X[09], 05, 16#21E1CDE6); (* 25 *)
	d := MD5_AUX(2, d, a, b, c, X[14], 09, 16#C33707D6); (* 26 *)
	c := MD5_AUX(2, c, d, a, b, X[03], 14, 16#F4D50D87); (* 27 *)
	b := MD5_AUX(2, b, c, d, a, X[08], 20, 16#455A14ED); (* 28 *)
	a := MD5_AUX(2, a, b, c, d, X[13], 05, 16#A9E3E905); (* 29 *)
	d := MD5_AUX(2, d, a, b, c, X[02], 09, 16#FCEFA3F8); (* 30 *)
	c := MD5_AUX(2, c, d, a, b, X[07], 14, 16#676F02D9); (* 31 *)
	b := MD5_AUX(2, b, c, d, a, X[12], 20, 16#8D2A4C8A); (* 32 *)

	a := MD5_AUX(3, a, b, c, d, X[05], 04, 16#FFFA3942); (* 33 *)
	d := MD5_AUX(3, d, a, b, c, X[08], 11, 16#8771F681); (* 34 *)
	c := MD5_AUX(3, c, d, a, b, X[11], 16, 16#6D9D6122); (* 35 *)
	b := MD5_AUX(3, b, c, d, a, X[14], 23, 16#FDE5380C); (* 36 *)
	a := MD5_AUX(3, a, b, c, d, X[01], 04, 16#A4BEEA44); (* 37 *)
	d := MD5_AUX(3, d, a, b, c, X[04], 11, 16#4BDECFA9); (* 38 *)
	c := MD5_AUX(3, c, d, a, b, X[07], 16, 16#F6BB4B60); (* 39 *)
	b := MD5_AUX(3, b, c, d, a, X[10], 23, 16#BEBFBC70); (* 40 *)
	a := MD5_AUX(3, a, b, c, d, X[13], 04, 16#289B7EC6); (* 41 *)
	d := MD5_AUX(3, d, a, b, c, X[00], 11, 16#EAA127FA); (* 42 *)
	c := MD5_AUX(3, c, d, a, b, X[03], 16, 16#D4EF3085); (* 43 *)
	b := MD5_AUX(3, b, c, d, a, X[06], 23, 16#04881D05); (* 44 *)
	a := MD5_AUX(3, a, b, c, d, X[09], 04, 16#D9D4D039); (* 45 *)
	d := MD5_AUX(3, d, a, b, c, X[12], 11, 16#E6DB99E5); (* 46 *)
	c := MD5_AUX(3, c, d, a, b, X[15], 16, 16#1FA27CF8); (* 47 *)
	b := MD5_AUX(3, b, c, d, a, X[02], 23, 16#C4AC5665); (* 48 *)

	a := MD5_AUX(4, a, b, c, d, X[00], 06, 16#F4292244); (* 49 *)
	d := MD5_AUX(4, d, a, b, c, X[07], 10, 16#432AFF97); (* 50 *)
	c := MD5_AUX(4, c, d, a, b, X[14], 15, 16#AB9423A7); (* 51 *)
	b := MD5_AUX(4, b, c, d, a, X[05], 21, 16#FC93A039); (* 52 *)
	a := MD5_AUX(4, a, b, c, d, X[12], 06, 16#655B59C3); (* 53 *)
	d := MD5_AUX(4, d, a, b, c, X[03], 10, 16#8F0CCC92); (* 54 *)
	c := MD5_AUX(4, c, d, a, b, X[10], 15, 16#FFEFF47D); (* 55 *)
	b := MD5_AUX(4, b, c, d, a, X[01], 21, 16#85845DD1); (* 56 *)
	a := MD5_AUX(4, a, b, c, d, X[08], 06, 16#6FA87E4F); (* 57 *)
	d := MD5_AUX(4, d, a, b, c, X[15], 10, 16#FE2CE6E0); (* 58 *)
	c := MD5_AUX(4, c, d, a, b, X[06], 15, 16#A3014314); (* 59 *)
	b := MD5_AUX(4, b, c, d, a, X[13], 21, 16#4E0811A1); (* 60 *)
	a := MD5_AUX(4, a, b, c, d, X[04], 06, 16#F7537E82); (* 61 *)
	d := MD5_AUX(4, d, a, b, c, X[11], 10, 16#BD3AF235); (* 62 *)
	c := MD5_AUX(4, c, d, a, b, X[02], 15, 16#2AD7D2BB); (* 63 *)
	b := MD5_AUX(4, b, c, d, a, X[09], 21, 16#EB86D391); (* 64 *)

	hash[0] := hash[0] + a;
	hash[1] := hash[1] + b;
	hash[2] := hash[2] + c;
	hash[3] := hash[3] + d;

END_CASE;

IF MODE = 3 THEN
	z := 0;
	FOR n := 0 TO 3 DO (* von Little-Endian auf Big-Endian format konvertieren und DWORD auf BYTE-Array *)
		FOR n1 := 0 TO 3 DO
			MD5[z] := DWORD_TO_BYTE(hash[n]);
			hash[n] := ROR(hash[n],8);
			z := z + 1;
		END_FOR;
	END_FOR;
END_IF;

(* revision history

ks	6. dec. 2009 rev 1.0
	original version

*)
END_FUNCTION_BLOCK

(* POU MD5_AUX, ST *)
FUNCTION MD5_AUX : DWORD
VAR_INPUT
	N : INT;
	A : DWORD;
	B : DWORD;
	C : DWORD;
	D : DWORD;
	X : DWORD;
	U : INT;
	T : DWORD;
END_VAR
VAR
	w : DWORD;
END_VAR

(*
version 1.0	06. dec. 2009
programmer 	ks
tested by	ks

MD5_AUX ist ein Zusatzbaustein füR MD5_STREAM und enthäLT wiederkehrende Berechnungen
*)
CASE N OF
	1: w := (B AND C) OR (NOT(B) AND D);
	2: w := (B AND D) OR (C AND NOT D);
	3: w := (B XOR C XOR D);
	4: w := (C XOR (B OR  NOT(D)));
END_CASE

MD5_AUX := B + ROL(A + w + X + T,U);

(* revision history

ks	6. dec. 2009 rev 1.0
	original version

*)
END_FUNCTION

(* POU MD5_TO_STRH, ST *)
FUNCTION MD5_TO_STRH : STRING(32)
VAR_INPUT
	MD5 : ARRAY [0..15] OF BYTE;
END_VAR
VAR
	i : INT;
	tmp : BYTE;
	pt : POINTER TO BYTE;
END_VAR
(*
version 1.0	06. dec. 2009
programmer 	ks
tested BY	ks

MD5_TO_STRH konvertiert das MD5 Hash Array in einen HEX-String
*)
pt := ADR(MD5_TO_STRH); (* read output adress to pointer *)

FOR i := 0 TO 15 DO; (* write the 8 hex characters backwards *)
	tmp := SHR(MD5[i],4);
	PT^ := tmp + SEL(tmp <= 9,87,48);
	pt := pt + 1; (* decrement the pointer *)
	tmp := MD5[i] AND 2#1111;
	PT^ := tmp + SEL(tmp <= 9,87,48);
	pt := pt + 1; (* decrement the pointer *)
END_FOR;
pt^:= 0; (* write the closing byte for the string *)

(* revision history

ks	6. dec. 2009 rev 1.0
	original version

*)
END_FUNCTION

(* POU ELEMENT_COUNT, ST *)
FUNCTION ELEMENT_COUNT : INT
VAR_INPUT
	SEP : BYTE;
END_VAR
VAR_IN_OUT
	ELEMENT : STRING(ELEMENT_LENGTH);
END_VAR
VAR
	pt : POINTER TO ARRAY[1..ELEMENT_LENGTH] OF BYTE;
	l: INT;
	pos: INT;
END_VAR

(*
version 1.0	05. apr. 2011
programmer 	hugo
tested by		oscat

ELEMENT_COUNT liefert die anzahl der elemente einer liste.
die liste liegt als string von elementen vor die mit den zeichen SEP separiert sind.

*)
IF ELEMENT = '' THEN
	ELEMENT_COUNT := 0;
ELSE
	PT := ADR(ELEMENT);
	ELEMENT_COUNT := 1;
	l := LEN(ELEMENT);
	FOR pos := 1 TO l DO
		IF pt^[pos] = SEP THEN ELEMENT_COUNT := ELEMENT_COUNT + 1; END_IF;
	END_FOR;
END_IF;

(* revision histroy
ks	5. apr. 2011	rev 1.0
	original release

*)	
END_FUNCTION

(* POU DLOG_RRD_DEMO, CFC *)
PROGRAM DLOG_RRD_DEMO
VAR
	RTC_2 : RTC_2;
	CLK_PRG: CLK_PRG;
	cur_dt : DT;
	rtc_set : BOOL := TRUE;
	enable : BOOL := TRUE;
	DLOG_STORE_RRD : DLOG_STORE_RRD;
	trig_t : UDINT := 0;
	trig_m : BOOL;

	rrd_done : BOOL;
	rrd_error_c : DWORD;
	rrd_error_t : BYTE;
	rrd_enable : BOOL := TRUE;
	rrd_url : STRING(STRING_LENGTH) := 'http://xxx.com/myhouse/rrd/test_rrd.php?rrd_db=test.rrd&value=';
	rrd_timeout: TIME := t#5s;

	x : DLOG_DATA;
	x1 : DLOG_DINT;
	x2 : DLOG_DINT;
	x3 : DLOG_REAL;
	x4 : DLOG_REAL;
	x5 : DLOG_REAL;
	x6 : DLOG_REAL;
	x7 : DLOG_REAL;

	GEN_SIN_1 : GEN_SIN;
	GEN_SIN_2 : GEN_SIN;
	GEN_SIN_3 : GEN_SIN;
	GEN_RMP_1: GEN_RMP;
	GEN_RMP_2: GEN_RMP;
END_VAR
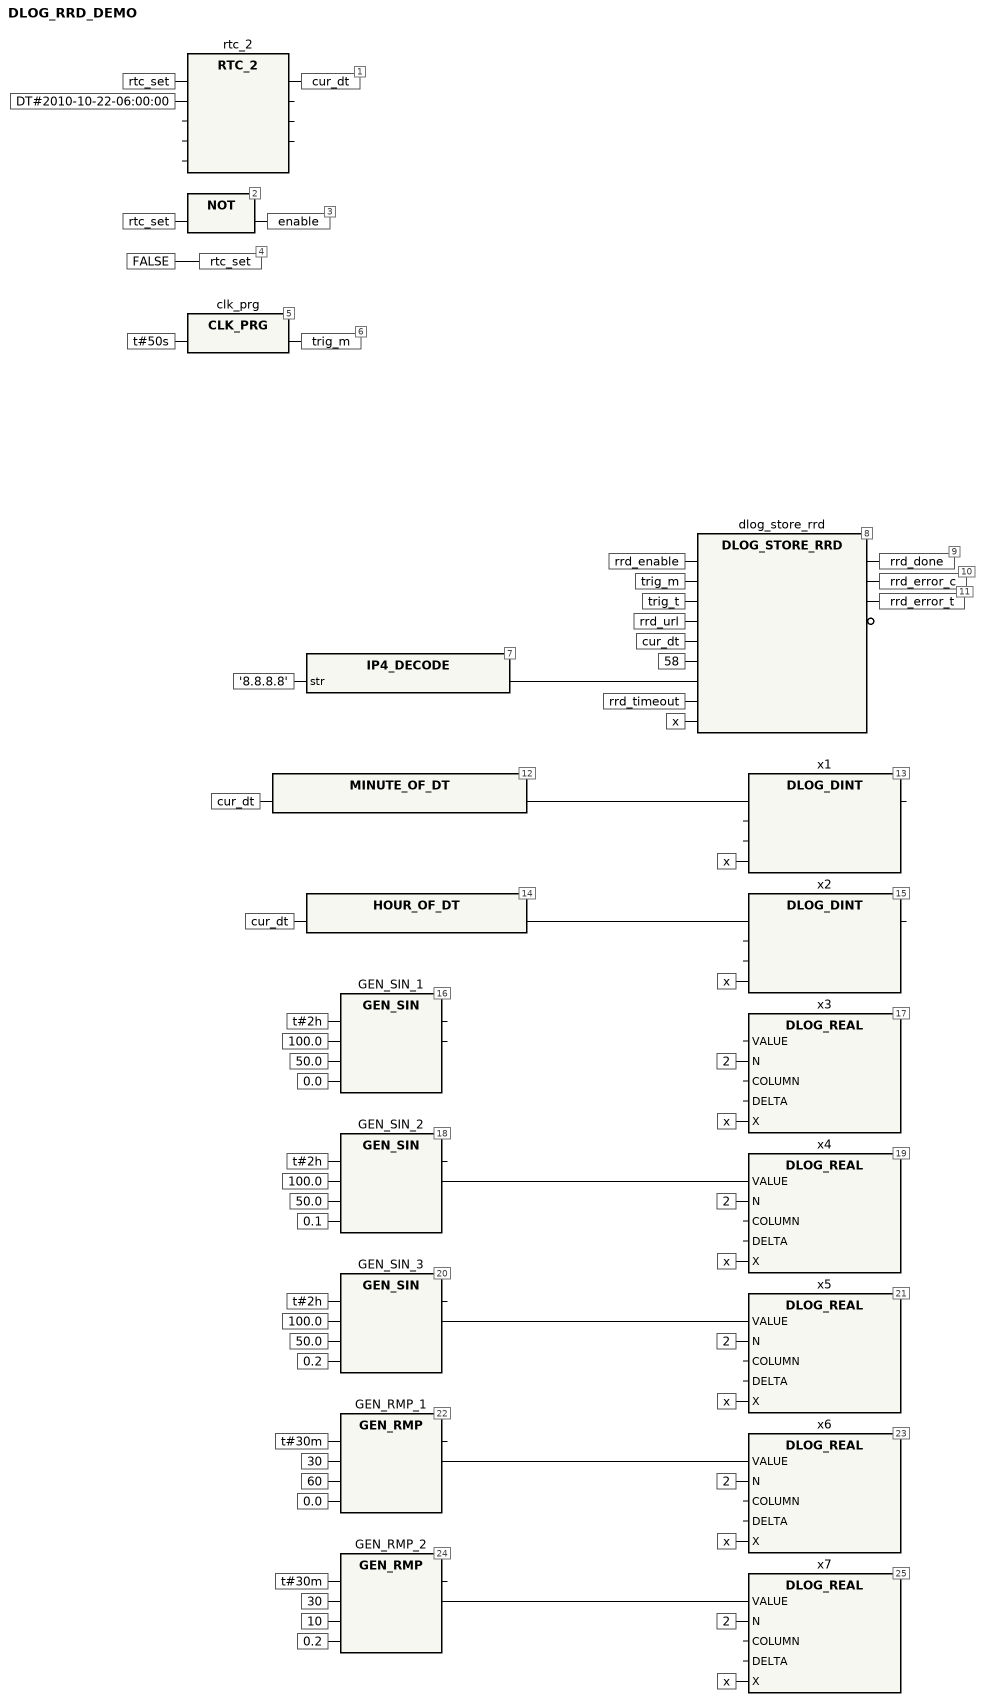
_CFC_ (* Continuous Function Chart, elements in execution order *)
#0 rtc_2:RTC_2(rtc_set, DT#2010-10-22-06:00:00, -, -, -)
#1 cur_dt <= #0.out 1
#2 NOT(rtc_set)
#3 enable <= #2
#4 rtc_set <= FALSE
#5 clk_prg:CLK_PRG(t#50s)
#6 trig_m <= #5
#7 IP4_DECODE(str: '8.8.8.8')
#8 dlog_store_rrd:DLOG_STORE_RRD(rrd_enable, trig_m, trig_t, rrd_url, cur_dt, 58, #7, rrd_timeout, x)
#9 rrd_done <= #8.out 1
#10 rrd_error_c <= #8.out 2
#11 rrd_error_t <= #8.out 3
#12 MINUTE_OF_DT(cur_dt)
#13 x1:DLOG_DINT(#12, -, -, x)
#14 HOUR_OF_DT(cur_dt)
#15 x2:DLOG_DINT(#14, -, -, x)
#16 GEN_SIN_1:GEN_SIN(t#2h, 100.0, 50.0, 0.0)
#17 x3:DLOG_REAL(VALUE: -, N: 2, COLUMN: -, DELTA: -, X: x)
#18 GEN_SIN_2:GEN_SIN(t#2h, 100.0, 50.0, 0.1)
#19 x4:DLOG_REAL(VALUE: #18.out 2, N: 2, COLUMN: -, DELTA: -, X: x)
#20 GEN_SIN_3:GEN_SIN(t#2h, 100.0, 50.0, 0.2)
#21 x5:DLOG_REAL(VALUE: #20.out 2, N: 2, COLUMN: -, DELTA: -, X: x)
#22 GEN_RMP_1:GEN_RMP(t#30m, 30, 60, 0.0)
#23 x6:DLOG_REAL(VALUE: #22.out 2, N: 2, COLUMN: -, DELTA: -, X: x)
#24 GEN_RMP_2:GEN_RMP(t#30m, 30, 10, 0.2)
#25 x7:DLOG_REAL(VALUE: #24.out 2, N: 2, COLUMN: -, DELTA: -, X: x)
_END_CFC_
END_PROGRAM

(* POU DLOG_STORE_RRD, ST *)
FUNCTION_BLOCK DLOG_STORE_RRD
VAR_IN_OUT
	X : DLOG_DATA;
END_VAR
VAR_INPUT
	ENABLE : BOOL;
	TRIG_M : BOOL;
	TRIG_T : UDINT;
	URL : STRING(STRING_LENGTH);
	DTI : DT;
	SEP : BYTE;
	DNS_IP4 : DWORD;
	TIMEOUT : TIME;
END_VAR
VAR_OUTPUT
	DONE : BOOL;
	ERROR_C : DWORD;
	ERROR_T : BYTE;
END_VAR
VAR
	UCB : UNI_CIRCULAR_BUFFER;
	IP_C : IP_C; (* IP_Control Verwaltungsstruktur *)
	S_BUF : NETWORK_BUFFER;
	R_BUF : NETWORK_BUFFER;
	URL_DATA : url;
	DNS_CLIENT : DNS_CLIENT;
	HTTP_GET : HTTP_GET;
	IPC : IP_CONTROL;

	ra : BOOL;
	trig_m_last : BOOL;
	dti_last : DT := DT#2070-02-06-06:28:15;
	enable_last : BOOL;
	step: INT;
	idx : INT;
	st1 : STRING(STRING_LENGTH);
	sep_char : STRING(1);
END_VAR

(*
version 1.1		13. may. 2011
programmer		ks
tested by			ks

DLOG_STORE_RRD der Baustein übergibt die DLOG Parameter an einen RoundRobinDatabase-Server
*)
X.DTI := DTI; (* Datum / Zeit eintragen *)
IF DTI <> dti_last THEN
	X.CLOCK_TRIG := TRUE;
	dti_last := DTI;
ELSE
	X.CLOCK_TRIG := FALSE;
END_IF;

X.ADD_DATA := FALSE;

IF ENABLE THEN
	IF X.CLOCK_TRIG THEN
		IF TRIG_T > 0 THEN (* automatischer Trigger *)
			ra := DT_TO_UDINT(DTI) MOD TRIG_T = 0;
		END_IF;
	ELSE
		ra := FALSE;
	END_IF;
	IF (TRIG_M AND NOT trig_m_last) OR ra OR X.ADD_DATA_REQ THEN (* manueller, automatischer oder externer Trigger *)
		X.ADD_DATA := TRUE; (* Daten loggen *)
	END_IF;
END_IF;
X.ADD_DATA_REQ := FALSE; (* externe Anforderung rücksetzen *)

CASE step OF

00:	IF ENABLE AND X.UCB.BUF_COUNT >= X.ID_MAX THEN (* mindestens eine ganze zeile im buffer *)
		sep_char := CHR_TO_STRING(SEP);
		DONE := FALSE;
		ERROR_T := 0;
		ERROR_C := 0;
		st1 := '';
		step := 20;
	END_IF;

20:	IF X.UCB.BUF_COUNT > 0 THEN (* Einträge vorhanden *)
		X.UCB.D_MODE := 10;
		UCB(DATA:=X.UCB); (* Element lesen , aber noch nicht entfernen *)
		IF LEN(st1) + LEN(X.UCB.D_STRING) + 1 <= STRING_LENGTH THEN
			st1 := CONCAT(st1,X.UCB.D_STRING);
		ELSE
			ERROR_T := 1; (* LOG-Daten können nicht in string gepackt werden *)
			ERROR_C := 1;
			step := 0;
		END_IF;
		X.UCB.D_MODE := 11;
		UCB(DATA:=X.UCB ); (* Element entfernen *)
		IF X.ID_MAX = SHR(X.UCB.D_HEAD,8) THEN (* letztes Element einer Zeile *)
			URL_DATA:=STRING_TO_URL(STR:=URL,DEFAULT_PROTOCOL:='',DEFAULT_PATH:=''); (* URL zerlegen *)
			IF LEN(st1) + LEN(URL_DATA.QUERY) <= 160 THEN
				URL_DATA.QUERY := CONCAT(URL_DATA.QUERY,st1); (* Query mit LOG-Daten ergänzen *)
				step :=40;
			ELSE
				ERROR_T := 4; (* LOG-Daten können nicht in URL gepackt werden *)
				ERROR_C := 1;
				step := 0;
			END_IF;
		ELSE
			st1 := CONCAT(st1,sep_char);
		END_IF;
	END_IF;

40:	IF DNS_CLIENT.DONE THEN
		step := 60;
	ELSIF (DNS_CLIENT.ERROR > 0) THEN
		ERROR_C := DNS_CLIENT.ERROR; (* Fehlerbehandlung *)
		ERROR_T := 1;
		step := 100;
	END_IF;

60:	IF HTTP_GET.DONE THEN
		idx := HTTP_GET.BODY_START;
		IF R_BUF.BUFFER[idx] = 48 THEN (* ASCII '0' *)
			DONE := TRUE;
		ELSE
			ERROR_C := 1;
			ERROR_T := 3;
		END_IF;
		step := 100;

	ELSIF HTTP_GET.ERROR > 0 THEN (* Fehlerbehandlung *)
		ERROR_C := HTTP_GET.ERROR;
		ERROR_T := 2;
		step := 100;
	END_IF;

100:	IF (NOT HTTP_GET.DONE) THEN (* UNLOCK HTTP DATA *)
		step := 0;
	END_IF;

END_CASE;

HTTP_GET(IP_C:=IP_C,S_BUF:=S_BUF,R_BUF:=R_BUF,IP4:=DNS_CLIENT.IP4,GET:=step=60,MODE:=2,UNLOCK_BUF:=step=100,URL_DATA:=URL_DATA); (* HTTP_GET *)
DNS_CLIENT(IP_C:=IP_C, S_BUF:=S_BUF, R_BUF:=R_BUF, DOMAIN:=URL_DATA.DOMAIN, IP4_DNS:= DNS_IP4, ACTIVATE:=step=40); (* DNS-Client *)
IPC(IP:= 0, PORT:= 0 , TIME_OUT:= TIMEOUT, IP_C:= IP_C, S_BUF:= S_BUF, R_BUF:= R_BUF); (* IP_CONTROL *)

trig_m_last := TRIG_M;
enable_last := ENABLE;

(* revision history
ks	01. jan. 2011	rev 1.0
	original version

ks	13. may. 2011	rev 1.1
	ADD_DATA_REQ hinzugefügt
*)
END_FUNCTION_BLOCK

(* POU HTTP_GET, ST *)
FUNCTION_BLOCK HTTP_GET
VAR_IN_OUT
	URL_DATA : url;
	IP_C : IP_C; (* IP_Control Verwaltungsstruktur *)
	S_BUF : NETWORK_BUFFER;
	R_BUF : NETWORK_BUFFER;
END_VAR
VAR_INPUT
	IP4 : DWORD;
	GET : BOOL;
	MODE : BYTE := BYTE#2;
	UNLOCK_BUF : BOOL;
END_VAR
VAR_OUTPUT
	HTTP_STATUS : STRING;
	HEADER_START : UINT; (* HTTP Header (Message Header) *)
	HEADER_STOP : UINT; (* HTTP Header (Message Header) *)
	BODY_START : UINT; (* Message Body *)
	BODY_STOP : UINT; (* Message Body *)
	DONE : BOOL;
	ERROR : DWORD;
END_VAR
VAR
	READ_HTTP :	READ_HTTP;
	IP_FIFO : IP_FIFO;
	ip_state : BYTE;
	ip_id : BYTE;
	get_last : BOOL;
	ip4_stored : DWORD;
	state : INT;
	i : INT;
	http_1_1_host : BOOL;
	total_size : INT;
	text : STRING(STRING_LENGTH);
	delimiter2b : STRING(2);
	delimiter4b : STRING(4);
	del_end : STRING(4);
	del_pos : INT;
	idx : INT;
	rcv_timeout : BOOL;
	con_rdce : BOOL;

	(*LOG_MSG : LOG_MSG;
	_debug_enable : BOOL := TRUE;*)

END_VAR

(*

version 1.3	12. apr. 2011
programmer 	ks
tested by		ks

HTTP_GET führt eine HTTP Abfrage einer Web-Seite bei einem WEB_Server durch, und stellt die Daten ausbereitet zu verfügung
*)
CASE state OF
00:	IF GET AND NOT GET_LAST THEN (* auf positive Flanke SET warten *)
		state := 10;
		ip4_stored := IP4; (* aktuelle IP4 speichern *)
		DONE := FALSE;
		total_size := 0;
		HEADER_START := UINT#0;
		HEADER_STOP := UINT#0;
		BODY_START := UINT#0;
		BODY_STOP := UINT#0;
		HTTP_STATUS := '';
		ERROR := DWORD#0;
		ip_state := BYTE#1; (* Anmelden *)
		delimiter2b := '$0D$0A';
		delimiter4b := '$0D$0A$0D$0A';
	        	(*####################  DEBUG-MESSAGE  ###################################*)
		(*IF _debug_enable THEN
	       		LOG_CL.NEW_MSG := 'HTTP: S00 START /IP_ID ~4';
	            	LOG_CL.PRINTF[4]  := BYTE_TO_STRING(IP_ID);
	            	LOG_MSG();
	        	END_IF;*)
	        	(*########################################################################*)
	END_IF;

10:	IF ip_state = BYTE#3 THEN (* Bei IP_Control anmelden und auf freigabe warten *)
		idx := 0;
		text := CONCAT('GET ',URL_DATA.PATH);
		_STRING_TO_BUFFER(STR:=text,POS:=idx,PT:=ADR(S_BUF.BUFFER),SIZE:=SIZEOF(S_BUF.BUFFER)); (* GET path in buffer kopieren *)
		idx := idx + LEN(text);

		IF LEN(URL_DATA.QUERY) > 0 THEN
			S_BUF.BUFFER[idx] := 63; (* ASCII '?' *)
			idx := idx + 1;
			_STRING_TO_BUFFER(STR:=URL_DATA.QUERY,POS:=idx,PT:=ADR(S_BUF.BUFFER),SIZE:=SIZEOF(S_BUF.BUFFER)); (* QUERY in buffer kopieren *)
			idx := idx + LEN(URL_DATA.QUERY);
		END_IF;

		IF MODE >= BYTE#2 THEN (* gewünschte HTTP Version uebergeben *)
			text := ' HTTP/1.1';
		ELSE
			text := ' HTTP/1.0';
		END_IF;
		text := CONCAT(text,delimiter2b);
		_STRING_TO_BUFFER(STR:=text,POS:=idx,PT:=ADR(S_BUF.BUFFER),SIZE:=SIZEOF(S_BUF.BUFFER)); (* HTTP Version in buffer kopieren *)
		idx := idx + LEN(text);

		IF MODE = BYTE#1 THEN (* HTTP/1.0 mit persistenter Verbindung gewünscht *)
			text := CONCAT('Connection: Keep-Alive',delimiter2b); (* workaround für pcworx -> kein $0D$0A als Stringkonstante möglich *)
		ELSIF MODE = BYTE#3 THEN (* HTTP/1.1 ohne persistenter Verbindung gewünscht *)
			text := CONCAT('Connection: Close',delimiter2b); (* workaround für pcworx -> kein $0D$0A als Stringkonstante möglich *)
		ELSE
			text := '';
		END_IF;
		text := CONCAT(text,URL_DATA.HEADER);
		_STRING_TO_BUFFER(STR:=text,POS:=idx,PT:=ADR(S_BUF.BUFFER),SIZE:=SIZEOF(S_BUF.BUFFER)); (* HTTP Version in buffer kopieren *)
		idx := idx + LEN(text);

		text := CONCAT('Host: ',URL_DATA.DOMAIN);
		text := CONCAT(text,delimiter4b); (* workaround für pcworx -> kein $0D$0A als Stringkonstante möglich *)
		_STRING_TO_BUFFER(STR:=text,POS:=idx,PT:=ADR(S_BUF.BUFFER),SIZE:=SIZEOF(S_BUF.BUFFER)); (* HTTP Host in buffer kopieren *)
		idx := idx + LEN(text);

		(* IP Datenverkehr einrichten *)
		IF URL_DATA.PORT = WORD#0 THEN
			IP_C.C_PORT := WORD#80; (* Standard-Portnummer verwenden *)
		ELSE
			IP_C.C_PORT := URL_DATA.PORT; (* Portnummer aus URL verwenden *)
		END_IF;

		IP_C.C_IP := ip4_stored; (* IP eintragen *)
		IP_C.C_MODE := BYTE#0; (* Mode: TCP+AKTIV+PORT+IP *)
		IP_C.C_ENABLE := TRUE; (* Verbindungsaufbau freigeben *)
		IP_C.TIME_RESET := TRUE; (* Zeitueberwachung rücksetzen *)
		IP_C.R_OBSERVE := TRUE; (* Datenempfang ueberwachen *)
		S_BUF.SIZE := INT_TO_UINT(idx); (* Sendelänge eintragen *)
		R_BUF.SIZE := UINT#0; (* Empfangslänge rücksetzen *)

		state := 30;
	        	(*####################  DEBUG-MESSAGE  ###################################*)
	        	(*IF _debug_enable THEN
	        		LOG_CL.NEW_MSG := 'HTTP: S20 SEND /IP_ID ~4';
	            	LOG_CL.PRINTF[4]  := BYTE_TO_STRING(IP_ID);
	            	LOG_MSG();
	        	END_IF;*)
	        	(*########################################################################*)
	END_IF;

30:	rcv_timeout := (IP_C.ERROR AND DWORD#16#0000_FF00) = DWORD#16#0000_FF00;
	con_rdce :=     (IP_C.ERROR AND DWORD#16#FD00_0000) = DWORD#16#FD00_0000;

	IF S_BUF.SIZE = UINT#0 THEN
		IF total_size = 0 THEN
			IF R_BUF.SIZE > UINT#15 THEN; (* länge der empfangenen Daten prüfen *)

				(* HTTP HEADER Ende suchen -> durch $0D$A$0D$A erkennbar bei DEC RT-11,CP/M,MS-DOS,Windows *)
				del_end := '$0D$0A$0D$0A';
				del_pos := BUFFER_SEARCH(PT:=ADR(R_BUF.BUFFER),SIZE:=R_BUF.SIZE,STR:=del_end,POS:=0,IGN:=FALSE);

				(* kein Ende gefunden ? -> andere Ende-Codierung suchen *)
				IF del_pos = 0 THEN
					del_end := '$0A$0A';
					(* HTTP HEADER Ende suchen -> durch $0A$0A erkennbar bei Multics, Unix-Derivate,Mac OS X *)
					del_pos := BUFFER_SEARCH(PT:=ADR(R_BUF.BUFFER),SIZE:=R_BUF.SIZE,STR:=del_end,POS:=0,IGN:=FALSE);
				END_IF;

				IF del_pos > 0 THEN
					HEADER_START := UINT#0;
					HEADER_STOP := INT_TO_UINT(del_pos + LEN(del_end) - 1);
					TOTAL_SIZE := -1; (* HTTP Header empfangen aber noch keine gesamtlänge bekannt *)
				END_IF;
		                	(*####################  DEBUG-MESSAGE  ###################################*)
		                	(*IF _debug_enable THEN
		                   	LOG_CL.NEW_MSG := 'HTTP: S20 HEADER_START ~1 / HEADER_STOP ~2/IP_ID ~4';
		                   	LOG_CL.PRINTF[4]  := BYTE_TO_STRING(IP_ID);
		                   	LOG_CL.PRINTF[1]  := UINT_TO_STRING(HEADER_START);
		                   	LOG_CL.PRINTF[2]  := UINT_TO_STRING(HEADER_STOP);
		                   	LOG_MSG();
		                	END_IF;*)
		                	(*########################################################################*)

				(* HTTP Statuscode auswerten: (kann 1.0 oder 1.1 sein *)
				READ_HTTP(size:=HEADER_STOP,pos:=0,SRC:='',pt:=R_BUF.BUFFER);

				i := LEN(READ_HTTP.READ_HTTP);
				IF i > 7 THEN
					(* HTTP Version von HOST auswerten 1.0 oder 1.1 *)
					text:=MID(READ_HTTP.READ_HTTP,1,3);
					http_1_1_host := text = '1';

					(* Code und Meldung isolieren *)
					HTTP_STATUS := RIGHT(READ_HTTP.READ_HTTP,i-4);
				END_IF;

				(* positive HTTP Anfrage ? *)
				IF FIND(HTTP_STATUS,'200') > 0 THEN

					(* 'Content-Length: Wert einlesen auswerten *)
					READ_HTTP(size:=HEADER_STOP,pos:=0,SRC:='CONTENT-LENGTH',pt:=R_BUF.BUFFER);
					text:=READ_HTTP.READ_HTTP;

					IF LEN(text) >= 1 THEN
						IF IS_NUM(str:=text) THEN
							(* erwartete gesamtmenge an Bytes berechnen *)
							total_size := STRING_TO_INT(text) + UINT_TO_INT(HEADER_STOP) + 1;
                           					(*####################  DEBUG-MESSAGE  ###################################*)
                           					(*IF _debug_enable THEN
                              					LOG_CL.NEW_MSG := 'HTTP: S20 HEADER ~1, BODY ~2 TOTAL ~3 /IP_ID ~4';
                             					LOG_CL.PRINTF[4]  := BYTE_TO_STRING(IP_ID);
                               					LOG_CL.PRINTF[1]  := UINT_TO_STRING(HEADER_STOP);
                               					LOG_CL.PRINTF[2]  := INT_TO_STRING(TOTAL_SIZE-UINT_TO_INT(HEADER_STOP));
                               					LOG_CL.PRINTF[3]  := INT_TO_STRING(TOTAL_SIZE);
                              					LOG_MSG();
                          					END_IF;*)
                          					(*########################################################################*)
						END_IF;
					END_IF;
				ELSE
					ERROR := DWORD#16#000000FC; (* Fehler durch HTTP-Statuscodes *)
				END_IF;
			END_IF;
		(* 1. bei bekannter Content-Length wird nach erhalt der erwartenen Daten die verbindung beendet *)
		(* 2. bei persistenter Verbindung muss bei unbekannter Datenmenge auf Receive-Timeout gewartet werden *)
		(* 3. wenn nach datenempfang die verbindung vom host unterbrochen wird *)
		ELSIF (R_BUF.SIZE >= INT_TO_UINT(total_size)) OR
			(R_BUF.SIZE > UINT#0 AND total_size < 0 AND ((rcv_timeout OR con_rdce) OR (IP_C.C_STATE = BYTE#1))) THEN

			IF R_BUF.SIZE - 1 > HEADER_STOP THEN (* BODY Daten vorhanden *)
				BODY_START := HEADER_STOP + UINT#1;
				BODY_STOP := R_BUF.SIZE - 1;
		                	(*####################  DEBUG-MESSAGE  ###################################*)
		                	(*IF _debug_enable THEN
		                   	LOG_CL.NEW_MSG := 'HTTP: S20 BODY ~1, START ~2 END ~3 /IP_ID ~4';
		                   	LOG_CL.PRINTF[4]  := BYTE_TO_STRING(IP_ID);
		                   	LOG_CL.PRINTF[1]  := UINT_TO_STRING(HEADER_STOP);
		                   	LOG_CL.PRINTF[2]  := UINT_TO_STRING(BODY_START);
		                   	LOG_CL.PRINTF[3]  := UINT_TO_STRING(BODY_STOP);
		                   	LOG_MSG();
		               	END_IF;*)
		               	(*########################################################################*)
			END_IF;

			DONE := TRUE;
			IP_C.C_ENABLE := FALSE; (* Verbindung abbauen *)
			state := 40;
            		(*####################  DEBUG-MESSAGE  ###################################*)
            		(*IF _debug_enable THEN
                			LOG_CL.NEW_MSG := 'HTTP: S30 OK /IP_ID ~4';
                			LOG_CL.PRINTF[4]  := BYTE_TO_STRING(IP_ID);
                			LOG_MSG();
            		END_IF;*)
            		(*########################################################################*)
		END_IF;
	END_IF;

	IF IP_C.ERROR <> DWORD#0 THEN
		(* bei unbekannter Content-size ist nicht bekannt ob bzw wieviele Telegramme noch folgen werden *)
		(* darum wird nach receive-timeout oder Remote disconnect error der fehler wieder ausgefiltert (logischer fehler) *)
		IF rcv_timeout AND DONE THEN
			IP_C.ERROR := IP_C.ERROR AND DWORD#16#FFFF_00FF; (* Fehler wieder rücksetzen *)
		ELSIF con_rdce AND DONE THEN
			IP_C.ERROR := IP_C.ERROR AND DWORD#16#00FF_FFFF; (* Fehler wieder rücksetzen *)
		ELSE
			ERROR := IP_C.ERROR;
		END_IF;
	END_IF;

	IF ERROR > DWORD#0 THEN
		IP_C.C_ENABLE := FALSE; (* Verbindungsaufbau sperren *)
		state := 40;
	        	(*####################  DEBUG-MESSAGE  ###################################*)
	        	(*IF _debug_enable THEN
	            	LOG_CL.NEW_MSG := 'HTTP: S30 ERROR ~1 /IP_ID ~4';
	            	LOG_CL.PRINTF[1]  := DWORD_TO_STRING(ERROR);
	            	LOG_CL.PRINTF[4]  := BYTE_TO_STRING(IP_ID);
	            	LOG_MSG();
	        	END_IF;*)
	        	(*########################################################################*)
	END_IF;

40:	IF (UNLOCK_BUF OR NOT DONE) THEN (* Warten auf Release und Verbindung beendet -> IP_ID vom Stack nehmen *)
		IP_STATE := BYTE#4; (* Abmelden *)
		DONE := FALSE;
		state := 0;
	END_IF;
END_CASE;

get_last := GET; (* letzten Status sichern zur Flankenerkennung *)

IP_FIFO(FIFO:=IP_C.FIFO,STATE:=ip_state,ID:=ip_id); (* IP_FIFO *)

(* revision history
ks	18. oct. 2008	rev 1.0
	original version

ks	20. oct. 2009	rev 1.1
	Fehler bei body-suche bei $0a$0a korrigiert,Codeoptimierung,
	new VAR del_pos , del_end (Networkbuffer und Buffer-funktionen auf Basis 0)

ks	28. oct. 2009	rev 1.2
	über url.header können zusätzliche header-infos übergeben werden

ks	12. apr. 2011	rev 1.3
	verbesserte fehlererkennung und fehlerkorrektur bei buffer_to_string
*)
END_FUNCTION_BLOCK

(* POU READ_HTTP, ST *)
FUNCTION_BLOCK READ_HTTP
VAR_INPUT
	SIZE : UINT;
	POS : INT;
	SRC : STRING;
END_VAR
VAR_IN_OUT
	PT : NW_BUF_LONG;
END_VAR
VAR_OUTPUT
	READ_HTTP : STRING(STRING_LENGTH);
END_VAR
VAR
	index : INT;
	s1 : INT;
	e1 : INT;
	stop : INT;
END_VAR

(*

version 1.1 20. oct. 2009
programmer 	ks
tested by	ks

READ_HTTP wertet die Informationen einer HTTP-Request aus, und stellt die Daten zu Verfügung.
*)
stop := UINT_TO_INT(SIZE) - 1;

IF LEN(SRC) = 0 THEN
	(* wenn kein Suchbegriff vorhanden ist, dann den HTTP-STATUS auswerten *)
	SRC := 'HTTP/'; (* neuer Suchbegriff *)
ELSE
	(* gesuchten Parametertext ergänzen *)
	SRC := CONCAT(SRC,': ');
END_IF;

s1 := BUFFER_SEARCH(pt:=ADR(PT),SIZE:=SIZE,STR:=SRC,POS:=POS,IGN:=TRUE);

IF s1 >= 0 THEN (* Text found *)
	e1 := s1;

	(* search start of line *)
	index := s1 - 1;
	WHILE (index > 0) DO
		IF pt[index] < BYTE#32 THEN EXIT; END_IF;
		s1 := s1 - 1;
		index := index - 1;
	END_WHILE;

	(* search end of line *)
	index := e1 + 1;
	WHILE (index <= stop) DO
		IF pt[index] < BYTE#32 THEN EXIT; END_IF;
		e1 := e1 + 1;
		index := index + 1;
	END_WHILE;

	s1 := s1 + LEN(SRC); (* 'suchbegriff: ' nicht mitkopieren *)

	(* copy string *)
	READ_HTTP := BUFFER_TO_STRING(PT:=ADR(PT),SIZE:=SIZE,START:=s1,STOP:=e1);
ELSE
	READ_HTTP := '';
END_IF;

(* revision history

ks	18. oct. 2008	rev 1.0
	original version

ks	20. oct. 2009	rev 1.1
	Networkbuffer und Buffer-funktionen auf Basis 0

*)
END_FUNCTION_BLOCK

(* POU DNS_DYN_DEMO, CFC *)
PROGRAM DNS_DYN_DEMO
VAR
	DNS_DYN : DNS_DYN;
	IP_C : IP_C;
	S_BUF : NETWORK_BUFFER;
	R_BUF : NETWORK_BUFFER;
	IP_CONTROL : IP_CONTROL;
	enable: BOOL;
	done : BOOL;
	error_c : DWORD;
	error_t : BYTE;
	busy : BOOL;
	COUNT_DR: COUNT_DR;
	z: DWORD;

